REGION Network 65: Transfer P&P Gague R&R Job Interface [Hipot & Thickness Loading][Right]
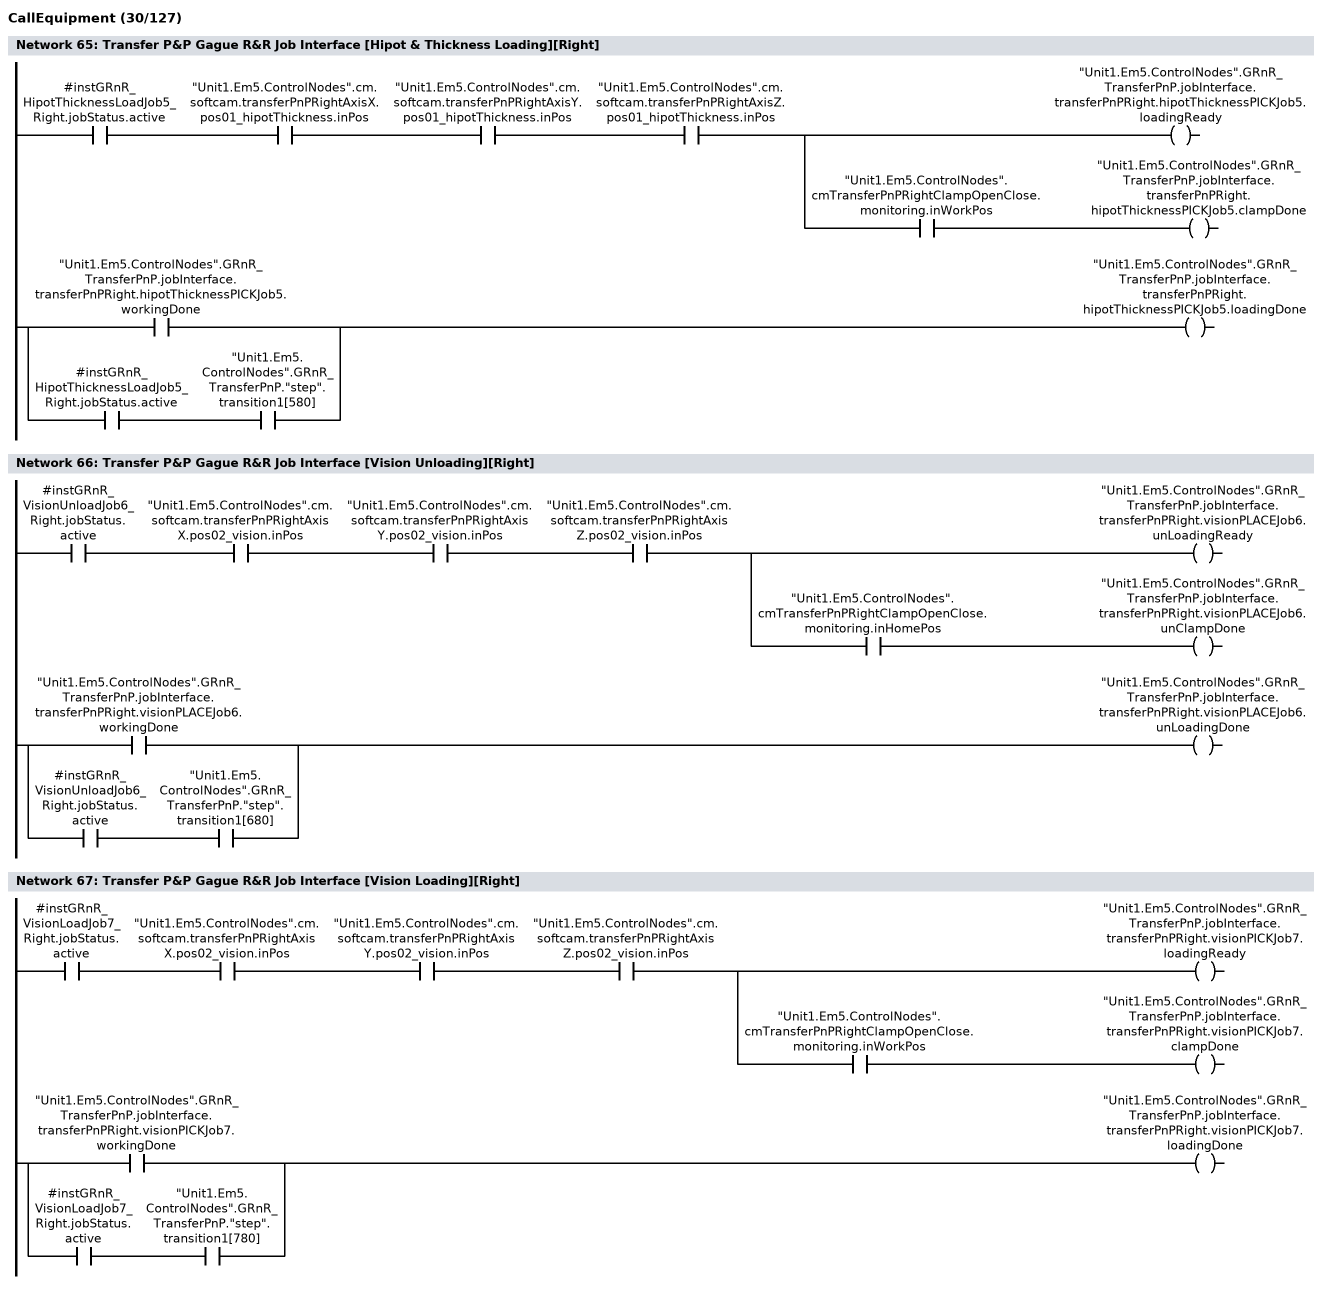
   RUNG wire#powerrail
      Contact( #instGRnR_HipotThicknessLoadJob5_Right.jobStatus.active )
      Contact( "Unit1.Em5.ControlNodes".cm.softcam.transferPnPRightAxisX.pos01_hipotThickness.inPos )
      Contact( "Unit1.Em5.ControlNodes".cm.softcam.transferPnPRightAxisY.pos01_hipotThickness.inPos )
      Contact( "Unit1.Em5.ControlNodes".cm.softcam.transferPnPRightAxisZ.pos01_hipotThickness.inPos )
      wire#w1
      Coil( "Unit1.Em5.ControlNodes".GRnR_TransferPnP.jobInterface.transferPnPRight.hipotThicknessPICKJob5.loadingReady )
   END_RUNG
   RUNG wire#w1
      Contact( "Unit1.Em5.ControlNodes".cmTransferPnPRightClampOpenClose.monitoring.inWorkPos )
      Coil( "Unit1.Em5.ControlNodes".GRnR_TransferPnP.jobInterface.transferPnPRight.hipotThicknessPICKJob5.clampDone )
   END_RUNG
   RUNG wire#powerrail
      Contact( "Unit1.Em5.ControlNodes".GRnR_TransferPnP.jobInterface.transferPnPRight.hipotThicknessPICKJob5.workingDone )
      wire#w2
      Coil( "Unit1.Em5.ControlNodes".GRnR_TransferPnP.jobInterface.transferPnPRight.hipotThicknessPICKJob5.loadingDone )
   END_RUNG
   RUNG wire#powerrail
      Contact( #instGRnR_HipotThicknessLoadJob5_Right.jobStatus.active )
      Contact( "Unit1.Em5.ControlNodes".GRnR_TransferPnP."step".transition1[580] )
   END_RUNG wire#w2
   // the same network as SCL:
   "Unit1.Em5.ControlNodes".GRnR_TransferPnP.jobInterface.transferPnPRight.hipotThicknessPICKJob5.loadingReady := #instGRnR_HipotThicknessLoadJob5_Right.jobStatus.active AND "Unit1.Em5.ControlNodes".cm.softcam.transferPnPRightAxisX.pos01_hipotThickness.inPos AND "Unit1.Em5.ControlNodes".cm.softcam.transferPnPRightAxisY.pos01_hipotThickness.inPos AND "Unit1.Em5.ControlNodes".cm.softcam.transferPnPRightAxisZ.pos01_hipotThickness.inPos;
   "Unit1.Em5.ControlNodes".GRnR_TransferPnP.jobInterface.transferPnPRight.hipotThicknessPICKJob5.clampDone := "Unit1.Em5.ControlNodes".GRnR_TransferPnP.jobInterface.transferPnPRight.hipotThicknessPICKJob5.loadingReady AND "Unit1.Em5.ControlNodes".cmTransferPnPRightClampOpenClose.monitoring.inWorkPos;
   "Unit1.Em5.ControlNodes".GRnR_TransferPnP.jobInterface.transferPnPRight.hipotThicknessPICKJob5.loadingDone := "Unit1.Em5.ControlNodes".GRnR_TransferPnP.jobInterface.transferPnPRight.hipotThicknessPICKJob5.workingDone OR (#instGRnR_HipotThicknessLoadJob5_Right.jobStatus.active AND "Unit1.Em5.ControlNodes".GRnR_TransferPnP."step".transition1[580]);
END_REGION

REGION Network 66: Transfer P&P Gague R&R Job Interface [Vision Unloading][Right]
   RUNG wire#powerrail
      Contact( #instGRnR_VisionUnloadJob6_Right.jobStatus.active )
      Contact( "Unit1.Em5.ControlNodes".cm.softcam.transferPnPRightAxisX.pos02_vision.inPos )
      Contact( "Unit1.Em5.ControlNodes".cm.softcam.transferPnPRightAxisY.pos02_vision.inPos )
      Contact( "Unit1.Em5.ControlNodes".cm.softcam.transferPnPRightAxisZ.pos02_vision.inPos )
      wire#w1
      Coil( "Unit1.Em5.ControlNodes".GRnR_TransferPnP.jobInterface.transferPnPRight.visionPLACEJob6.unLoadingReady )
   END_RUNG
   RUNG wire#w1
      Contact( "Unit1.Em5.ControlNodes".cmTransferPnPRightClampOpenClose.monitoring.inHomePos )
      Coil( "Unit1.Em5.ControlNodes".GRnR_TransferPnP.jobInterface.transferPnPRight.visionPLACEJob6.unClampDone )
   END_RUNG
   RUNG wire#powerrail
      Contact( "Unit1.Em5.ControlNodes".GRnR_TransferPnP.jobInterface.transferPnPRight.visionPLACEJob6.workingDone )
      wire#w2
      Coil( "Unit1.Em5.ControlNodes".GRnR_TransferPnP.jobInterface.transferPnPRight.visionPLACEJob6.unLoadingDone )
   END_RUNG
   RUNG wire#powerrail
      Contact( #instGRnR_VisionUnloadJob6_Right.jobStatus.active )
      Contact( "Unit1.Em5.ControlNodes".GRnR_TransferPnP."step".transition1[680] )
   END_RUNG wire#w2
   // the same network as SCL:
   "Unit1.Em5.ControlNodes".GRnR_TransferPnP.jobInterface.transferPnPRight.visionPLACEJob6.unLoadingReady := #instGRnR_VisionUnloadJob6_Right.jobStatus.active AND "Unit1.Em5.ControlNodes".cm.softcam.transferPnPRightAxisX.pos02_vision.inPos AND "Unit1.Em5.ControlNodes".cm.softcam.transferPnPRightAxisY.pos02_vision.inPos AND "Unit1.Em5.ControlNodes".cm.softcam.transferPnPRightAxisZ.pos02_vision.inPos;
   "Unit1.Em5.ControlNodes".GRnR_TransferPnP.jobInterface.transferPnPRight.visionPLACEJob6.unClampDone := "Unit1.Em5.ControlNodes".GRnR_TransferPnP.jobInterface.transferPnPRight.visionPLACEJob6.unLoadingReady AND "Unit1.Em5.ControlNodes".cmTransferPnPRightClampOpenClose.monitoring.inHomePos;
   "Unit1.Em5.ControlNodes".GRnR_TransferPnP.jobInterface.transferPnPRight.visionPLACEJob6.unLoadingDone := "Unit1.Em5.ControlNodes".GRnR_TransferPnP.jobInterface.transferPnPRight.visionPLACEJob6.workingDone OR (#instGRnR_VisionUnloadJob6_Right.jobStatus.active AND "Unit1.Em5.ControlNodes".GRnR_TransferPnP."step".transition1[680]);
END_REGION

REGION Network 67: Transfer P&P Gague R&R Job Interface [Vision Loading][Right]
   RUNG wire#powerrail
      Contact( #instGRnR_VisionLoadJob7_Right.jobStatus.active )
      Contact( "Unit1.Em5.ControlNodes".cm.softcam.transferPnPRightAxisX.pos02_vision.inPos )
      Contact( "Unit1.Em5.ControlNodes".cm.softcam.transferPnPRightAxisY.pos02_vision.inPos )
      Contact( "Unit1.Em5.ControlNodes".cm.softcam.transferPnPRightAxisZ.pos02_vision.inPos )
      wire#w1
      Coil( "Unit1.Em5.ControlNodes".GRnR_TransferPnP.jobInterface.transferPnPRight.visionPICKJob7.loadingReady )
   END_RUNG
   RUNG wire#w1
      Contact( "Unit1.Em5.ControlNodes".cmTransferPnPRightClampOpenClose.monitoring.inWorkPos )
      Coil( "Unit1.Em5.ControlNodes".GRnR_TransferPnP.jobInterface.transferPnPRight.visionPICKJob7.clampDone )
   END_RUNG
   RUNG wire#powerrail
      Contact( "Unit1.Em5.ControlNodes".GRnR_TransferPnP.jobInterface.transferPnPRight.visionPICKJob7.workingDone )
      wire#w2
      Coil( "Unit1.Em5.ControlNodes".GRnR_TransferPnP.jobInterface.transferPnPRight.visionPICKJob7.loadingDone )
   END_RUNG
   RUNG wire#powerrail
      Contact( #instGRnR_VisionLoadJob7_Right.jobStatus.active )
      Contact( "Unit1.Em5.ControlNodes".GRnR_TransferPnP."step".transition1[780] )
   END_RUNG wire#w2
   // the same network as SCL:
   "Unit1.Em5.ControlNodes".GRnR_TransferPnP.jobInterface.transferPnPRight.visionPICKJob7.loadingReady := #instGRnR_VisionLoadJob7_Right.jobStatus.active AND "Unit1.Em5.ControlNodes".cm.softcam.transferPnPRightAxisX.pos02_vision.inPos AND "Unit1.Em5.ControlNodes".cm.softcam.transferPnPRightAxisY.pos02_vision.inPos AND "Unit1.Em5.ControlNodes".cm.softcam.transferPnPRightAxisZ.pos02_vision.inPos;
   "Unit1.Em5.ControlNodes".GRnR_TransferPnP.jobInterface.transferPnPRight.visionPICKJob7.clampDone := "Unit1.Em5.ControlNodes".GRnR_TransferPnP.jobInterface.transferPnPRight.visionPICKJob7.loadingReady AND "Unit1.Em5.ControlNodes".cmTransferPnPRightClampOpenClose.monitoring.inWorkPos;
   "Unit1.Em5.ControlNodes".GRnR_TransferPnP.jobInterface.transferPnPRight.visionPICKJob7.loadingDone := "Unit1.Em5.ControlNodes".GRnR_TransferPnP.jobInterface.transferPnPRight.visionPICKJob7.workingDone OR (#instGRnR_VisionLoadJob7_Right.jobStatus.active AND "Unit1.Em5.ControlNodes".GRnR_TransferPnP."step".transition1[780]);
END_REGION

REGION Network 68: Transfer P&P Gague R&R Job Interface [Weight Check Unloading][Right]
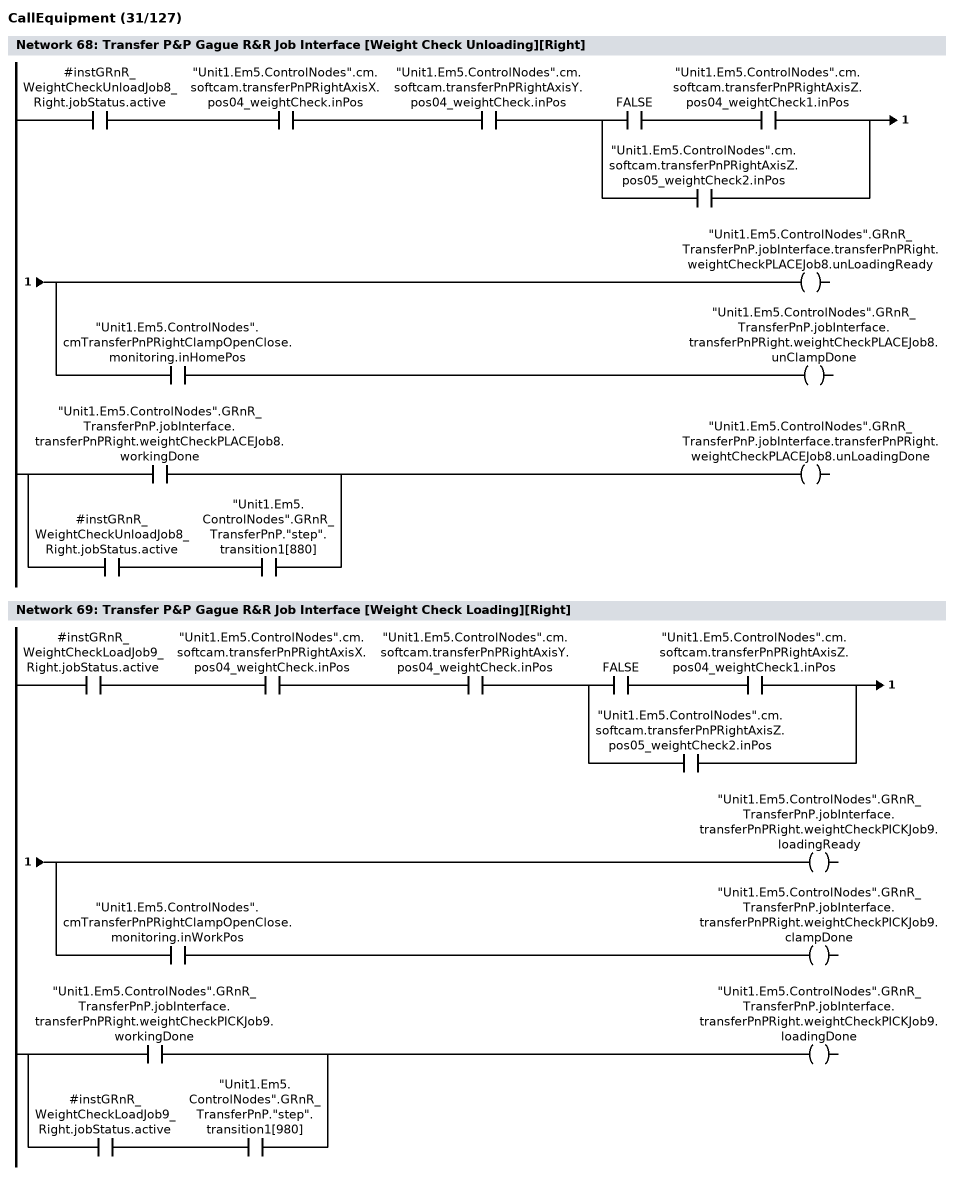
   RUNG wire#powerrail
      Contact( #instGRnR_WeightCheckUnloadJob8_Right.jobStatus.active )
      Contact( "Unit1.Em5.ControlNodes".cm.softcam.transferPnPRightAxisX.pos04_weightCheck.inPos )
      Contact( "Unit1.Em5.ControlNodes".cm.softcam.transferPnPRightAxisY.pos04_weightCheck.inPos )
      wire#w1
      Contact( FALSE )
      Contact( "Unit1.Em5.ControlNodes".cm.softcam.transferPnPRightAxisZ.pos04_weightCheck1.inPos )
      wire#w2
      Coil( "Unit1.Em5.ControlNodes".GRnR_TransferPnP.jobInterface.transferPnPRight.weightCheckPLACEJob8.unLoadingReady )
   END_RUNG
   RUNG wire#w1
      Contact( "Unit1.Em5.ControlNodes".cm.softcam.transferPnPRightAxisZ.pos05_weightCheck2.inPos )
   END_RUNG wire#w2
   RUNG wire#w2
      Contact( "Unit1.Em5.ControlNodes".cmTransferPnPRightClampOpenClose.monitoring.inHomePos )
      Coil( "Unit1.Em5.ControlNodes".GRnR_TransferPnP.jobInterface.transferPnPRight.weightCheckPLACEJob8.unClampDone )
   END_RUNG
   RUNG wire#powerrail
      Contact( "Unit1.Em5.ControlNodes".GRnR_TransferPnP.jobInterface.transferPnPRight.weightCheckPLACEJob8.workingDone )
      wire#w3
      Coil( "Unit1.Em5.ControlNodes".GRnR_TransferPnP.jobInterface.transferPnPRight.weightCheckPLACEJob8.unLoadingDone )
   END_RUNG
   RUNG wire#powerrail
      Contact( #instGRnR_WeightCheckUnloadJob8_Right.jobStatus.active )
      Contact( "Unit1.Em5.ControlNodes".GRnR_TransferPnP."step".transition1[880] )
   END_RUNG wire#w3
   // the same network as SCL:
   "Unit1.Em5.ControlNodes".GRnR_TransferPnP.jobInterface.transferPnPRight.weightCheckPLACEJob8.unLoadingReady := #instGRnR_WeightCheckUnloadJob8_Right.jobStatus.active AND "Unit1.Em5.ControlNodes".cm.softcam.transferPnPRightAxisX.pos04_weightCheck.inPos AND "Unit1.Em5.ControlNodes".cm.softcam.transferPnPRightAxisY.pos04_weightCheck.inPos AND ((FALSE AND "Unit1.Em5.ControlNodes".cm.softcam.transferPnPRightAxisZ.pos04_weightCheck1.inPos) OR "Unit1.Em5.ControlNodes".cm.softcam.transferPnPRightAxisZ.pos05_weightCheck2.inPos);
   "Unit1.Em5.ControlNodes".GRnR_TransferPnP.jobInterface.transferPnPRight.weightCheckPLACEJob8.unClampDone := "Unit1.Em5.ControlNodes".GRnR_TransferPnP.jobInterface.transferPnPRight.weightCheckPLACEJob8.unLoadingReady AND "Unit1.Em5.ControlNodes".cmTransferPnPRightClampOpenClose.monitoring.inHomePos;
   "Unit1.Em5.ControlNodes".GRnR_TransferPnP.jobInterface.transferPnPRight.weightCheckPLACEJob8.unLoadingDone := "Unit1.Em5.ControlNodes".GRnR_TransferPnP.jobInterface.transferPnPRight.weightCheckPLACEJob8.workingDone OR (#instGRnR_WeightCheckUnloadJob8_Right.jobStatus.active AND "Unit1.Em5.ControlNodes".GRnR_TransferPnP."step".transition1[880]);
END_REGION

REGION Network 69: Transfer P&P Gague R&R Job Interface [Weight Check Loading][Right]
   RUNG wire#powerrail
      Contact( #instGRnR_WeightCheckLoadJob9_Right.jobStatus.active )
      Contact( "Unit1.Em5.ControlNodes".cm.softcam.transferPnPRightAxisX.pos04_weightCheck.inPos )
      Contact( "Unit1.Em5.ControlNodes".cm.softcam.transferPnPRightAxisY.pos04_weightCheck.inPos )
      wire#w1
      Contact( FALSE )
      Contact( "Unit1.Em5.ControlNodes".cm.softcam.transferPnPRightAxisZ.pos04_weightCheck1.inPos )
      wire#w2
      Coil( "Unit1.Em5.ControlNodes".GRnR_TransferPnP.jobInterface.transferPnPRight.weightCheckPICKJob9.loadingReady )
   END_RUNG
   RUNG wire#w1
      Contact( "Unit1.Em5.ControlNodes".cm.softcam.transferPnPRightAxisZ.pos05_weightCheck2.inPos )
   END_RUNG wire#w2
   RUNG wire#w2
      Contact( "Unit1.Em5.ControlNodes".cmTransferPnPRightClampOpenClose.monitoring.inWorkPos )
      Coil( "Unit1.Em5.ControlNodes".GRnR_TransferPnP.jobInterface.transferPnPRight.weightCheckPICKJob9.clampDone )
   END_RUNG
   RUNG wire#powerrail
      Contact( "Unit1.Em5.ControlNodes".GRnR_TransferPnP.jobInterface.transferPnPRight.weightCheckPICKJob9.workingDone )
      wire#w3
      Coil( "Unit1.Em5.ControlNodes".GRnR_TransferPnP.jobInterface.transferPnPRight.weightCheckPICKJob9.loadingDone )
   END_RUNG
   RUNG wire#powerrail
      Contact( #instGRnR_WeightCheckLoadJob9_Right.jobStatus.active )
      Contact( "Unit1.Em5.ControlNodes".GRnR_TransferPnP."step".transition1[980] )
   END_RUNG wire#w3
   // the same network as SCL:
   "Unit1.Em5.ControlNodes".GRnR_TransferPnP.jobInterface.transferPnPRight.weightCheckPICKJob9.loadingReady := #instGRnR_WeightCheckLoadJob9_Right.jobStatus.active AND "Unit1.Em5.ControlNodes".cm.softcam.transferPnPRightAxisX.pos04_weightCheck.inPos AND "Unit1.Em5.ControlNodes".cm.softcam.transferPnPRightAxisY.pos04_weightCheck.inPos AND ((FALSE AND "Unit1.Em5.ControlNodes".cm.softcam.transferPnPRightAxisZ.pos04_weightCheck1.inPos) OR "Unit1.Em5.ControlNodes".cm.softcam.transferPnPRightAxisZ.pos05_weightCheck2.inPos);
   "Unit1.Em5.ControlNodes".GRnR_TransferPnP.jobInterface.transferPnPRight.weightCheckPICKJob9.clampDone := "Unit1.Em5.ControlNodes".GRnR_TransferPnP.jobInterface.transferPnPRight.weightCheckPICKJob9.loadingReady AND "Unit1.Em5.ControlNodes".cmTransferPnPRightClampOpenClose.monitoring.inWorkPos;
   "Unit1.Em5.ControlNodes".GRnR_TransferPnP.jobInterface.transferPnPRight.weightCheckPICKJob9.loadingDone := "Unit1.Em5.ControlNodes".GRnR_TransferPnP.jobInterface.transferPnPRight.weightCheckPICKJob9.workingDone OR (#instGRnR_WeightCheckLoadJob9_Right.jobStatus.active AND "Unit1.Em5.ControlNodes".GRnR_TransferPnP."step".transition1[980]);
END_REGION

REGION Network 70: Transfer P&P Gague R&R Job Interface Working Done [Side Tape → Hipot & Thickness]
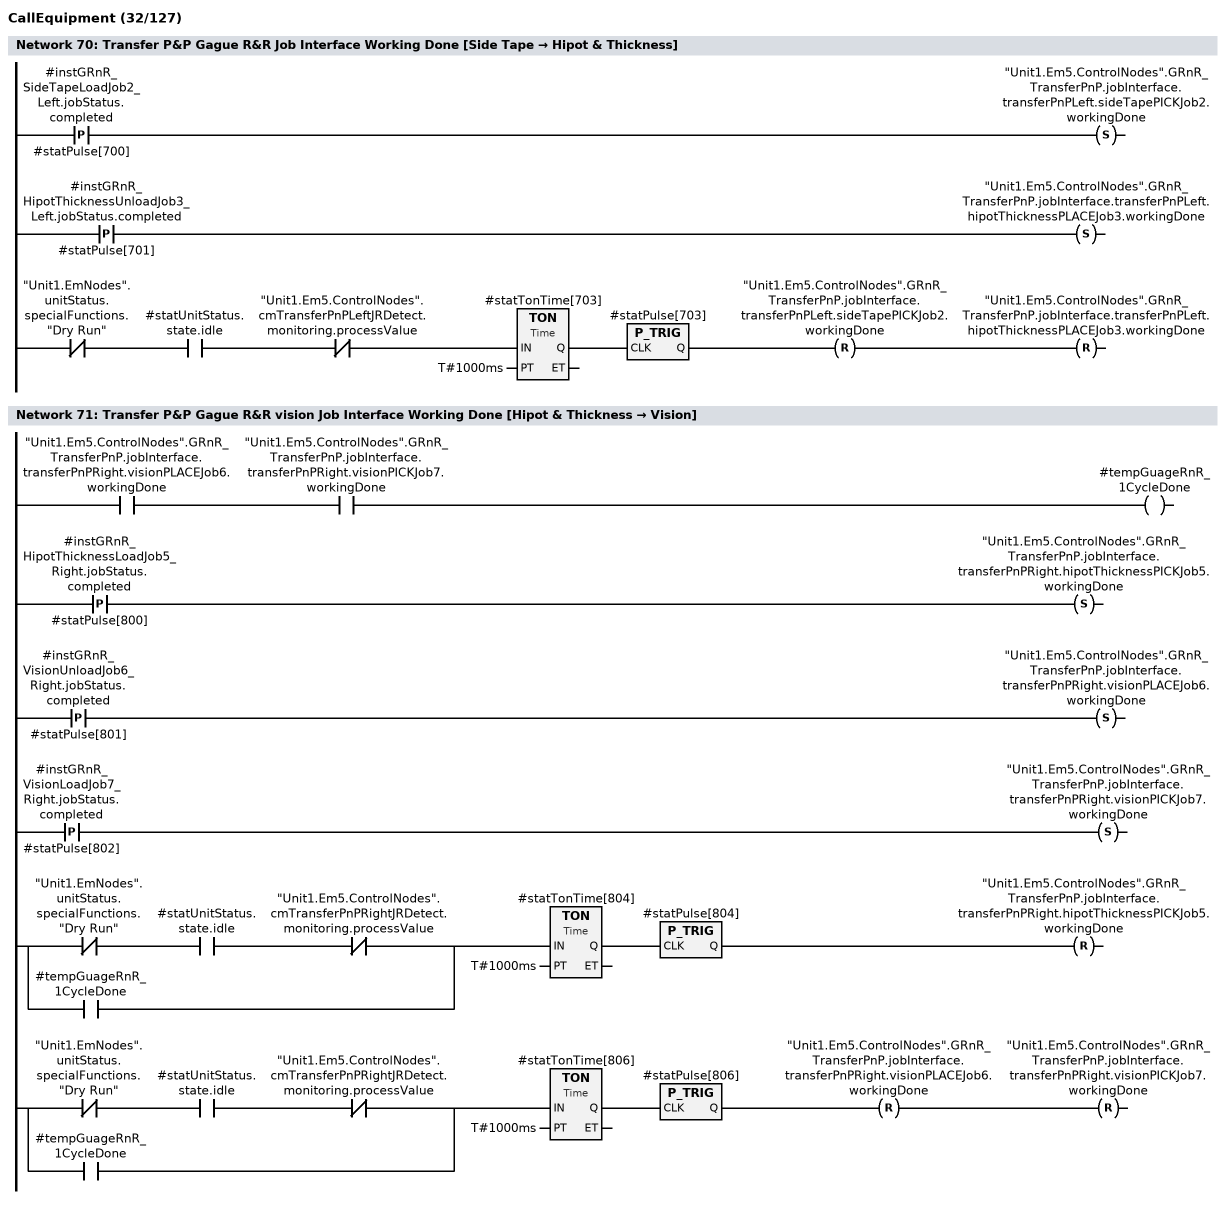
   RUNG wire#powerrail
      P_Contact(operand := #instGRnR_SideTapeLoadJob2_Left.jobStatus.completed, bit := #statPulse[700])
      S_Coil( "Unit1.Em5.ControlNodes".GRnR_TransferPnP.jobInterface.transferPnPLeft.sideTapePICKJob2.workingDone )
   END_RUNG
   RUNG wire#powerrail
      P_Contact(operand := #instGRnR_HipotThicknessUnloadJob3_Left.jobStatus.completed, bit := #statPulse[701])
      S_Coil( "Unit1.Em5.ControlNodes".GRnR_TransferPnP.jobInterface.transferPnPLeft.hipotThicknessPLACEJob3.workingDone )
   END_RUNG
   RUNG wire#powerrail
      I_Contact( "Unit1.EmNodes".unitStatus.specialFunctions."Dry Run" )
      Contact( #statUnitStatus.state.idle )
      I_Contact( "Unit1.Em5.ControlNodes".cmTransferPnPLeftJRDetect.monitoring.processValue )
      { S7_Templates := "time_type := Time" } #statTonTime[703].TON(pt := T#1000ms, et =>)
      P_Trig( #statPulse[703] )
      R_Coil( "Unit1.Em5.ControlNodes".GRnR_TransferPnP.jobInterface.transferPnPLeft.sideTapePICKJob2.workingDone )
      R_Coil( "Unit1.Em5.ControlNodes".GRnR_TransferPnP.jobInterface.transferPnPLeft.hipotThicknessPLACEJob3.workingDone )
   END_RUNG
   // the same network as SCL:
   #_w1 := #instGRnR_SideTapeLoadJob2_Left.jobStatus.completed AND NOT #statPulse[700];   // rising edge of #instGRnR_SideTapeLoadJob2_Left.jobStatus.completed
   #statPulse[700] := #instGRnR_SideTapeLoadJob2_Left.jobStatus.completed;
   IF #_w1 THEN
       "Unit1.Em5.ControlNodes".GRnR_TransferPnP.jobInterface.transferPnPLeft.sideTapePICKJob2.workingDone := TRUE;
   END_IF;
   #_w2 := #instGRnR_HipotThicknessUnloadJob3_Left.jobStatus.completed AND NOT #statPulse[701];   // rising edge of #instGRnR_HipotThicknessUnloadJob3_Left.jobStatus.completed
   #statPulse[701] := #instGRnR_HipotThicknessUnloadJob3_Left.jobStatus.completed;
   IF #_w2 THEN
       "Unit1.Em5.ControlNodes".GRnR_TransferPnP.jobInterface.transferPnPLeft.hipotThicknessPLACEJob3.workingDone := TRUE;
   END_IF;
   #statTonTime[703].TON(IN := NOT "Unit1.EmNodes".unitStatus.specialFunctions."Dry Run" AND #statUnitStatus.state.idle AND NOT "Unit1.Em5.ControlNodes".cmTransferPnPLeftJRDetect.monitoring.processValue,
                         PT := T#1000ms);
   #_w3 := #statTonTime[703].Q AND NOT #statPulse[703];   // rising edge
   #statPulse[703] := #statTonTime[703].Q;
   IF #_w3 THEN
       "Unit1.Em5.ControlNodes".GRnR_TransferPnP.jobInterface.transferPnPLeft.sideTapePICKJob2.workingDone := FALSE;
       "Unit1.Em5.ControlNodes".GRnR_TransferPnP.jobInterface.transferPnPLeft.hipotThicknessPLACEJob3.workingDone := FALSE;
   END_IF;
END_REGION

REGION Network 71: Transfer P&P Gague R&R vision Job Interface Working Done [Hipot & Thickness → Vision]
   RUNG wire#powerrail
      Contact( "Unit1.Em5.ControlNodes".GRnR_TransferPnP.jobInterface.transferPnPRight.visionPLACEJob6.workingDone )
      Contact( "Unit1.Em5.ControlNodes".GRnR_TransferPnP.jobInterface.transferPnPRight.visionPICKJob7.workingDone )
      Coil( #tempGuageRnR_1CycleDone )
   END_RUNG
   RUNG wire#powerrail
      P_Contact(operand := #instGRnR_HipotThicknessLoadJob5_Right.jobStatus.completed, bit := #statPulse[800])
      S_Coil( "Unit1.Em5.ControlNodes".GRnR_TransferPnP.jobInterface.transferPnPRight.hipotThicknessPICKJob5.workingDone )
   END_RUNG
   RUNG wire#powerrail
      P_Contact(operand := #instGRnR_VisionUnloadJob6_Right.jobStatus.completed, bit := #statPulse[801])
      S_Coil( "Unit1.Em5.ControlNodes".GRnR_TransferPnP.jobInterface.transferPnPRight.visionPLACEJob6.workingDone )
   END_RUNG
   RUNG wire#powerrail
      P_Contact(operand := #instGRnR_VisionLoadJob7_Right.jobStatus.completed, bit := #statPulse[802])
      S_Coil( "Unit1.Em5.ControlNodes".GRnR_TransferPnP.jobInterface.transferPnPRight.visionPICKJob7.workingDone )
   END_RUNG
   RUNG wire#powerrail
      I_Contact( "Unit1.EmNodes".unitStatus.specialFunctions."Dry Run" )
      Contact( #statUnitStatus.state.idle )
      I_Contact( "Unit1.Em5.ControlNodes".cmTransferPnPRightJRDetect.monitoring.processValue )
      wire#w1
      { S7_Templates := "time_type := Time" } #statTonTime[804].TON(pt := T#1000ms, et =>)
      P_Trig( #statPulse[804] )
      R_Coil( "Unit1.Em5.ControlNodes".GRnR_TransferPnP.jobInterface.transferPnPRight.hipotThicknessPICKJob5.workingDone )
   END_RUNG
   RUNG wire#powerrail
      Contact( #tempGuageRnR_1CycleDone )
   END_RUNG wire#w1
   RUNG wire#powerrail
      I_Contact( "Unit1.EmNodes".unitStatus.specialFunctions."Dry Run" )
      Contact( #statUnitStatus.state.idle )
      I_Contact( "Unit1.Em5.ControlNodes".cmTransferPnPRightJRDetect.monitoring.processValue )
      wire#w2
      { S7_Templates := "time_type := Time" } #statTonTime[806].TON(pt := T#1000ms, et =>)
      P_Trig( #statPulse[806] )
      R_Coil( "Unit1.Em5.ControlNodes".GRnR_TransferPnP.jobInterface.transferPnPRight.visionPLACEJob6.workingDone )
      R_Coil( "Unit1.Em5.ControlNodes".GRnR_TransferPnP.jobInterface.transferPnPRight.visionPICKJob7.workingDone )
   END_RUNG
   RUNG wire#powerrail
      Contact( #tempGuageRnR_1CycleDone )
   END_RUNG wire#w2
   // the same network as SCL:
   #tempGuageRnR_1CycleDone := "Unit1.Em5.ControlNodes".GRnR_TransferPnP.jobInterface.transferPnPRight.visionPLACEJob6.workingDone AND "Unit1.Em5.ControlNodes".GRnR_TransferPnP.jobInterface.transferPnPRight.visionPICKJob7.workingDone;
   #_w1 := #instGRnR_HipotThicknessLoadJob5_Right.jobStatus.completed AND NOT #statPulse[800];   // rising edge of #instGRnR_HipotThicknessLoadJob5_Right.jobStatus.completed
   #statPulse[800] := #instGRnR_HipotThicknessLoadJob5_Right.jobStatus.completed;
   IF #_w1 THEN
       "Unit1.Em5.ControlNodes".GRnR_TransferPnP.jobInterface.transferPnPRight.hipotThicknessPICKJob5.workingDone := TRUE;
   END_IF;
   #_w2 := #instGRnR_VisionUnloadJob6_Right.jobStatus.completed AND NOT #statPulse[801];   // rising edge of #instGRnR_VisionUnloadJob6_Right.jobStatus.completed
   #statPulse[801] := #instGRnR_VisionUnloadJob6_Right.jobStatus.completed;
   IF #_w2 THEN
       "Unit1.Em5.ControlNodes".GRnR_TransferPnP.jobInterface.transferPnPRight.visionPLACEJob6.workingDone := TRUE;
   END_IF;
   #_w3 := #instGRnR_VisionLoadJob7_Right.jobStatus.completed AND NOT #statPulse[802];   // rising edge of #instGRnR_VisionLoadJob7_Right.jobStatus.completed
   #statPulse[802] := #instGRnR_VisionLoadJob7_Right.jobStatus.completed;
   IF #_w3 THEN
       "Unit1.Em5.ControlNodes".GRnR_TransferPnP.jobInterface.transferPnPRight.visionPICKJob7.workingDone := TRUE;
   END_IF;
   #statTonTime[804].TON(IN := (NOT "Unit1.EmNodes".unitStatus.specialFunctions."Dry Run" AND #statUnitStatus.state.idle AND NOT "Unit1.Em5.ControlNodes".cmTransferPnPRightJRDetect.monitoring.processValue) OR #tempGuageRnR_1CycleDone,
                         PT := T#1000ms);
   #_w4 := #statTonTime[804].Q AND NOT #statPulse[804];   // rising edge
   #statPulse[804] := #statTonTime[804].Q;
   IF #_w4 THEN
       "Unit1.Em5.ControlNodes".GRnR_TransferPnP.jobInterface.transferPnPRight.hipotThicknessPICKJob5.workingDone := FALSE;
   END_IF;
   #statTonTime[806].TON(IN := (NOT "Unit1.EmNodes".unitStatus.specialFunctions."Dry Run" AND #statUnitStatus.state.idle AND NOT "Unit1.Em5.ControlNodes".cmTransferPnPRightJRDetect.monitoring.processValue) OR #tempGuageRnR_1CycleDone,
                         PT := T#1000ms);
   #_w5 := #statTonTime[806].Q AND NOT #statPulse[806];   // rising edge
   #statPulse[806] := #statTonTime[806].Q;
   IF #_w5 THEN
       "Unit1.Em5.ControlNodes".GRnR_TransferPnP.jobInterface.transferPnPRight.visionPLACEJob6.workingDone := FALSE;
       "Unit1.Em5.ControlNodes".GRnR_TransferPnP.jobInterface.transferPnPRight.visionPICKJob7.workingDone := FALSE;
   END_IF;
END_REGION

REGION Network 72: Transfer P&P Gague R&R Job Interface Working Done [Vision → Weight Check]
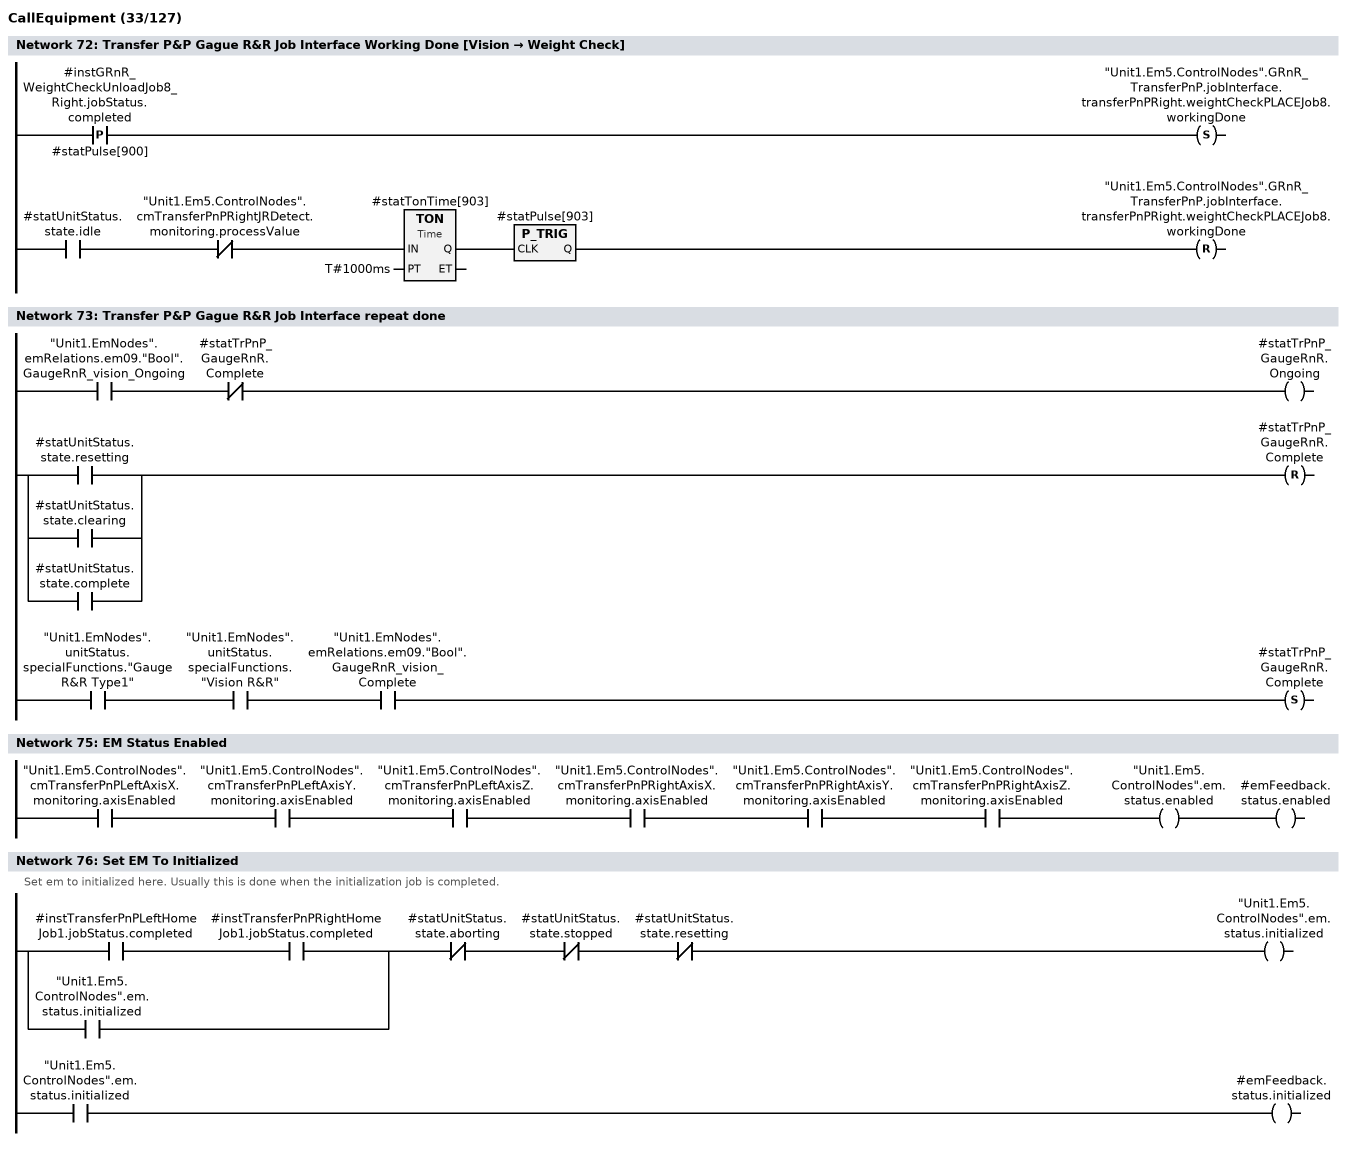
   RUNG wire#powerrail
      P_Contact(operand := #instGRnR_WeightCheckUnloadJob8_Right.jobStatus.completed, bit := #statPulse[900])
      S_Coil( "Unit1.Em5.ControlNodes".GRnR_TransferPnP.jobInterface.transferPnPRight.weightCheckPLACEJob8.workingDone )
   END_RUNG
   RUNG wire#powerrail
      Contact( #statUnitStatus.state.idle )
      I_Contact( "Unit1.Em5.ControlNodes".cmTransferPnPRightJRDetect.monitoring.processValue )
      { S7_Templates := "time_type := Time" } #statTonTime[903].TON(pt := T#1000ms, et =>)
      P_Trig( #statPulse[903] )
      R_Coil( "Unit1.Em5.ControlNodes".GRnR_TransferPnP.jobInterface.transferPnPRight.weightCheckPLACEJob8.workingDone )
   END_RUNG
   // the same network as SCL:
   #_w1 := #instGRnR_WeightCheckUnloadJob8_Right.jobStatus.completed AND NOT #statPulse[900];   // rising edge of #instGRnR_WeightCheckUnloadJob8_Right.jobStatus.completed
   #statPulse[900] := #instGRnR_WeightCheckUnloadJob8_Right.jobStatus.completed;
   IF #_w1 THEN
       "Unit1.Em5.ControlNodes".GRnR_TransferPnP.jobInterface.transferPnPRight.weightCheckPLACEJob8.workingDone := TRUE;
   END_IF;
   #statTonTime[903].TON(IN := #statUnitStatus.state.idle AND NOT "Unit1.Em5.ControlNodes".cmTransferPnPRightJRDetect.monitoring.processValue,
                         PT := T#1000ms);
   #_w2 := #statTonTime[903].Q AND NOT #statPulse[903];   // rising edge
   #statPulse[903] := #statTonTime[903].Q;
   IF #_w2 THEN
       "Unit1.Em5.ControlNodes".GRnR_TransferPnP.jobInterface.transferPnPRight.weightCheckPLACEJob8.workingDone := FALSE;
   END_IF;
END_REGION

REGION Network 73: Transfer P&P Gague R&R Job Interface repeat done
   RUNG wire#powerrail
      Contact( "Unit1.EmNodes".emRelations.em09."Bool".GaugeRnR_vision_Ongoing )
      I_Contact( #statTrPnP_GaugeRnR.Complete )
      Coil( #statTrPnP_GaugeRnR.Ongoing )
   END_RUNG
   RUNG wire#powerrail
      Contact( #statUnitStatus.state.resetting )
      wire#w1
      R_Coil( #statTrPnP_GaugeRnR.Complete )
   END_RUNG
   RUNG wire#powerrail
      Contact( #statUnitStatus.state.clearing )
   END_RUNG wire#w1
   RUNG wire#powerrail
      Contact( #statUnitStatus.state.complete )
   END_RUNG wire#w1
   RUNG wire#powerrail
      Contact( "Unit1.EmNodes".unitStatus.specialFunctions."Gauge R&R Type1" )
      Contact( "Unit1.EmNodes".unitStatus.specialFunctions."Vision R&R" )
      Contact( "Unit1.EmNodes".emRelations.em09."Bool".GaugeRnR_vision_Complete )
      S_Coil( #statTrPnP_GaugeRnR.Complete )
   END_RUNG
   // the same network as SCL:
   #statTrPnP_GaugeRnR.Ongoing := "Unit1.EmNodes".emRelations.em09."Bool".GaugeRnR_vision_Ongoing AND NOT #statTrPnP_GaugeRnR.Complete;
   IF #statUnitStatus.state.resetting OR #statUnitStatus.state.clearing OR #statUnitStatus.state.complete THEN
       #statTrPnP_GaugeRnR.Complete := FALSE;
   END_IF;
   IF "Unit1.EmNodes".unitStatus.specialFunctions."Gauge R&R Type1" AND "Unit1.EmNodes".unitStatus.specialFunctions."Vision R&R" AND "Unit1.EmNodes".emRelations.em09."Bool".GaugeRnR_vision_Complete THEN
       #statTrPnP_GaugeRnR.Complete := TRUE;
   END_IF;
END_REGION

REGION Network 75: EM Status Enabled
   RUNG wire#powerrail
      Contact( "Unit1.Em5.ControlNodes".cmTransferPnPLeftAxisX.monitoring.axisEnabled )
      Contact( "Unit1.Em5.ControlNodes".cmTransferPnPLeftAxisY.monitoring.axisEnabled )
      Contact( "Unit1.Em5.ControlNodes".cmTransferPnPLeftAxisZ.monitoring.axisEnabled )
      Contact( "Unit1.Em5.ControlNodes".cmTransferPnPRightAxisX.monitoring.axisEnabled )
      Contact( "Unit1.Em5.ControlNodes".cmTransferPnPRightAxisY.monitoring.axisEnabled )
      Contact( "Unit1.Em5.ControlNodes".cmTransferPnPRightAxisZ.monitoring.axisEnabled )
      Coil( "Unit1.Em5.ControlNodes".em.status.enabled )
      Coil( #emFeedback.status.enabled )
   END_RUNG
   // the same network as SCL:
   "Unit1.Em5.ControlNodes".em.status.enabled := "Unit1.Em5.ControlNodes".cmTransferPnPLeftAxisX.monitoring.axisEnabled AND "Unit1.Em5.ControlNodes".cmTransferPnPLeftAxisY.monitoring.axisEnabled AND "Unit1.Em5.ControlNodes".cmTransferPnPLeftAxisZ.monitoring.axisEnabled AND "Unit1.Em5.ControlNodes".cmTransferPnPRightAxisX.monitoring.axisEnabled AND "Unit1.Em5.ControlNodes".cmTransferPnPRightAxisY.monitoring.axisEnabled AND "Unit1.Em5.ControlNodes".cmTransferPnPRightAxisZ.monitoring.axisEnabled;
   #emFeedback.status.enabled := "Unit1.Em5.ControlNodes".em.status.enabled;
END_REGION

REGION Network 76: Set EM To Initialized
   // Set em to initialized here. Usually this is done when the initialization job is completed.
   RUNG wire#powerrail
      Contact( #instTransferPnPLeftHomeJob1.jobStatus.completed )
      Contact( #instTransferPnPRightHomeJob1.jobStatus.completed )
      wire#w1
      I_Contact( #statUnitStatus.state.aborting )
      I_Contact( #statUnitStatus.state.stopped )
      I_Contact( #statUnitStatus.state.resetting )
      Coil( "Unit1.Em5.ControlNodes".em.status.initialized )
   END_RUNG
   RUNG wire#powerrail
      Contact( "Unit1.Em5.ControlNodes".em.status.initialized )
   END_RUNG wire#w1
   RUNG wire#powerrail
      Contact( "Unit1.Em5.ControlNodes".em.status.initialized )
      Coil( #emFeedback.status.initialized )
   END_RUNG
   // the same network as SCL:
   "Unit1.Em5.ControlNodes".em.status.initialized := ((#instTransferPnPLeftHomeJob1.jobStatus.completed AND #instTransferPnPRightHomeJob1.jobStatus.completed) OR "Unit1.Em5.ControlNodes".em.status.initialized) AND NOT #statUnitStatus.state.aborting AND NOT #statUnitStatus.state.stopped AND NOT #statUnitStatus.state.resetting;
   #emFeedback.status.initialized := "Unit1.Em5.ControlNodes".em.status.initialized;
END_REGION

REGION Network 77: EM Status Homed
   // DefaultPosPartDetect : TR PnP Right has a Part, and no where to go
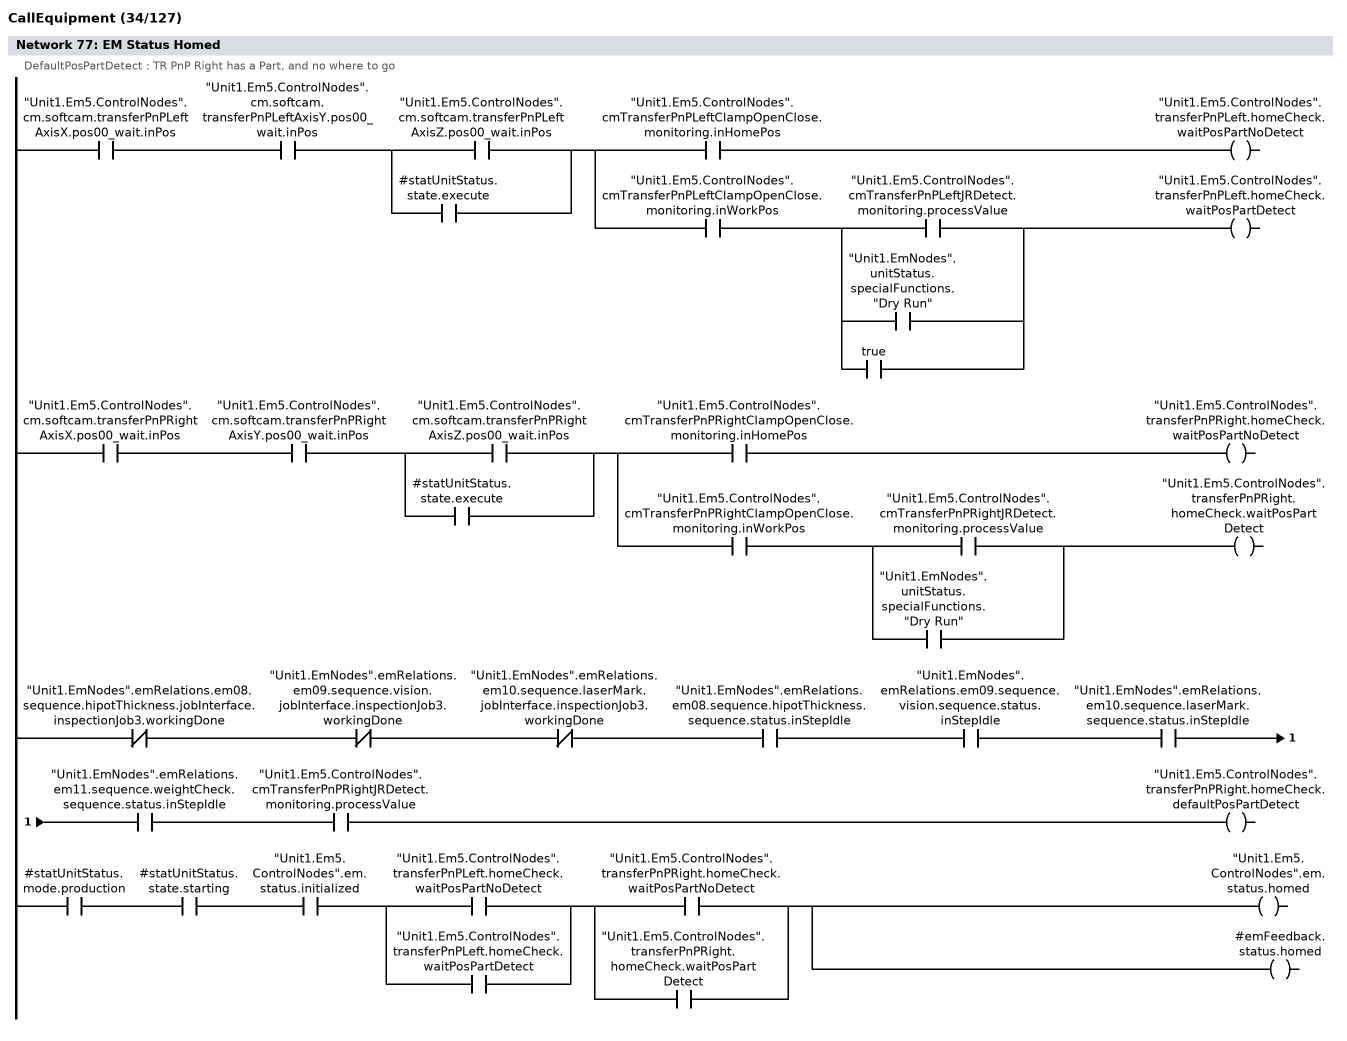
   RUNG wire#powerrail
      Contact( "Unit1.Em5.ControlNodes".cm.softcam.transferPnPLeftAxisX.pos00_wait.inPos )
      Contact( "Unit1.Em5.ControlNodes".cm.softcam.transferPnPLeftAxisY.pos00_wait.inPos )
      wire#w1
      Contact( "Unit1.Em5.ControlNodes".cm.softcam.transferPnPLeftAxisZ.pos00_wait.inPos )
      wire#w2
      Contact( "Unit1.Em5.ControlNodes".cmTransferPnPLeftClampOpenClose.monitoring.inHomePos )
      Coil( "Unit1.Em5.ControlNodes".transferPnPLeft.homeCheck.waitPosPartNoDetect )
   END_RUNG
   RUNG wire#w1
      Contact( #statUnitStatus.state.execute )
   END_RUNG wire#w2
   RUNG wire#w2
      Contact( "Unit1.Em5.ControlNodes".cmTransferPnPLeftClampOpenClose.monitoring.inWorkPos )
      wire#w3
      Contact( "Unit1.Em5.ControlNodes".cmTransferPnPLeftJRDetect.monitoring.processValue )
      wire#w4
      Coil( "Unit1.Em5.ControlNodes".transferPnPLeft.homeCheck.waitPosPartDetect )
   END_RUNG
   RUNG wire#w3
      Contact( "Unit1.EmNodes".unitStatus.specialFunctions."Dry Run" )
   END_RUNG wire#w4
   RUNG wire#w3
      Contact( true )
   END_RUNG wire#w4
   RUNG wire#powerrail
      Contact( "Unit1.Em5.ControlNodes".cm.softcam.transferPnPRightAxisX.pos00_wait.inPos )
      Contact( "Unit1.Em5.ControlNodes".cm.softcam.transferPnPRightAxisY.pos00_wait.inPos )
      wire#w5
      Contact( "Unit1.Em5.ControlNodes".cm.softcam.transferPnPRightAxisZ.pos00_wait.inPos )
      wire#w6
      Contact( "Unit1.Em5.ControlNodes".cmTransferPnPRightClampOpenClose.monitoring.inHomePos )
      Coil( "Unit1.Em5.ControlNodes".transferPnPRight.homeCheck.waitPosPartNoDetect )
   END_RUNG
   RUNG wire#w5
      Contact( #statUnitStatus.state.execute )
   END_RUNG wire#w6
   RUNG wire#w6
      Contact( "Unit1.Em5.ControlNodes".cmTransferPnPRightClampOpenClose.monitoring.inWorkPos )
      wire#w7
      Contact( "Unit1.Em5.ControlNodes".cmTransferPnPRightJRDetect.monitoring.processValue )
      wire#w8
      Coil( "Unit1.Em5.ControlNodes".transferPnPRight.homeCheck.waitPosPartDetect )
   END_RUNG
   RUNG wire#w7
      Contact( "Unit1.EmNodes".unitStatus.specialFunctions."Dry Run" )
   END_RUNG wire#w8
   RUNG wire#powerrail
      I_Contact( "Unit1.EmNodes".emRelations.em08.sequence.hipotThickness.jobInterface.inspectionJob3.workingDone )
      I_Contact( "Unit1.EmNodes".emRelations.em09.sequence.vision.jobInterface.inspectionJob3.workingDone )
      I_Contact( "Unit1.EmNodes".emRelations.em10.sequence.laserMark.jobInterface.inspectionJob3.workingDone )
      Contact( "Unit1.EmNodes".emRelations.em08.sequence.hipotThickness.sequence.status.inStepIdle )
      Contact( "Unit1.EmNodes".emRelations.em09.sequence.vision.sequence.status.inStepIdle )
      Contact( "Unit1.EmNodes".emRelations.em10.sequence.laserMark.sequence.status.inStepIdle )
      Contact( "Unit1.EmNodes".emRelations.em11.sequence.weightCheck.sequence.status.inStepIdle )
      Contact( "Unit1.Em5.ControlNodes".cmTransferPnPRightJRDetect.monitoring.processValue )
      Coil( "Unit1.Em5.ControlNodes".transferPnPRight.homeCheck.defaultPosPartDetect )
   END_RUNG
   RUNG wire#powerrail
      Contact( #statUnitStatus.mode.production )
      Contact( #statUnitStatus.state.starting )
      Contact( "Unit1.Em5.ControlNodes".em.status.initialized )
      wire#w9
      Contact( "Unit1.Em5.ControlNodes".transferPnPLeft.homeCheck.waitPosPartNoDetect )
      wire#w10
      Contact( "Unit1.Em5.ControlNodes".transferPnPRight.homeCheck.waitPosPartNoDetect )
      wire#w11
      Coil( "Unit1.Em5.ControlNodes".em.status.homed )
   END_RUNG
   RUNG wire#w9
      Contact( "Unit1.Em5.ControlNodes".transferPnPLeft.homeCheck.waitPosPartDetect )
   END_RUNG wire#w10
   RUNG wire#w10
      Contact( "Unit1.Em5.ControlNodes".transferPnPRight.homeCheck.waitPosPartDetect )
   END_RUNG wire#w11
   RUNG wire#w11
      Coil( #emFeedback.status.homed )
   END_RUNG
   // the same network as SCL:
   #_w1 := "Unit1.Em5.ControlNodes".cm.softcam.transferPnPLeftAxisX.pos00_wait.inPos AND "Unit1.Em5.ControlNodes".cm.softcam.transferPnPLeftAxisY.pos00_wait.inPos AND ("Unit1.Em5.ControlNodes".cm.softcam.transferPnPLeftAxisZ.pos00_wait.inPos OR #statUnitStatus.state.execute);
   "Unit1.Em5.ControlNodes".transferPnPLeft.homeCheck.waitPosPartNoDetect := #_w1 AND "Unit1.Em5.ControlNodes".cmTransferPnPLeftClampOpenClose.monitoring.inHomePos;
   "Unit1.Em5.ControlNodes".transferPnPLeft.homeCheck.waitPosPartDetect := #_w1 AND "Unit1.Em5.ControlNodes".cmTransferPnPLeftClampOpenClose.monitoring.inWorkPos AND ("Unit1.Em5.ControlNodes".cmTransferPnPLeftJRDetect.monitoring.processValue OR "Unit1.EmNodes".unitStatus.specialFunctions."Dry Run" OR true);
   #_w2 := "Unit1.Em5.ControlNodes".cm.softcam.transferPnPRightAxisX.pos00_wait.inPos AND "Unit1.Em5.ControlNodes".cm.softcam.transferPnPRightAxisY.pos00_wait.inPos AND ("Unit1.Em5.ControlNodes".cm.softcam.transferPnPRightAxisZ.pos00_wait.inPos OR #statUnitStatus.state.execute);
   "Unit1.Em5.ControlNodes".transferPnPRight.homeCheck.waitPosPartNoDetect := #_w2 AND "Unit1.Em5.ControlNodes".cmTransferPnPRightClampOpenClose.monitoring.inHomePos;
   "Unit1.Em5.ControlNodes".transferPnPRight.homeCheck.waitPosPartDetect := #_w2 AND "Unit1.Em5.ControlNodes".cmTransferPnPRightClampOpenClose.monitoring.inWorkPos AND ("Unit1.Em5.ControlNodes".cmTransferPnPRightJRDetect.monitoring.processValue OR "Unit1.EmNodes".unitStatus.specialFunctions."Dry Run");
   "Unit1.Em5.ControlNodes".transferPnPRight.homeCheck.defaultPosPartDetect := NOT "Unit1.EmNodes".emRelations.em08.sequence.hipotThickness.jobInterface.inspectionJob3.workingDone AND NOT "Unit1.EmNodes".emRelations.em09.sequence.vision.jobInterface.inspectionJob3.workingDone AND NOT "Unit1.EmNodes".emRelations.em10.sequence.laserMark.jobInterface.inspectionJob3.workingDone AND "Unit1.EmNodes".emRelations.em08.sequence.hipotThickness.sequence.status.inStepIdle AND "Unit1.EmNodes".emRelations.em09.sequence.vision.sequence.status.inStepIdle AND "Unit1.EmNodes".emRelations.em10.sequence.laserMark.sequence.status.inStepIdle AND "Unit1.EmNodes".emRelations.em11.sequence.weightCheck.sequence.status.inStepIdle AND "Unit1.Em5.ControlNodes".cmTransferPnPRightJRDetect.monitoring.processValue;
   "Unit1.Em5.ControlNodes".em.status.homed := #statUnitStatus.mode.production AND #statUnitStatus.state.starting AND "Unit1.Em5.ControlNodes".em.status.initialized AND ("Unit1.Em5.ControlNodes".transferPnPLeft.homeCheck.waitPosPartNoDetect OR "Unit1.Em5.ControlNodes".transferPnPLeft.homeCheck.waitPosPartDetect) AND ("Unit1.Em5.ControlNodes".transferPnPRight.homeCheck.waitPosPartNoDetect OR "Unit1.Em5.ControlNodes".transferPnPRight.homeCheck.waitPosPartDetect);
   #emFeedback.status.homed := "Unit1.Em5.ControlNodes".em.status.homed;
END_REGION

REGION Network 78: Transfer P&P Left Position Check
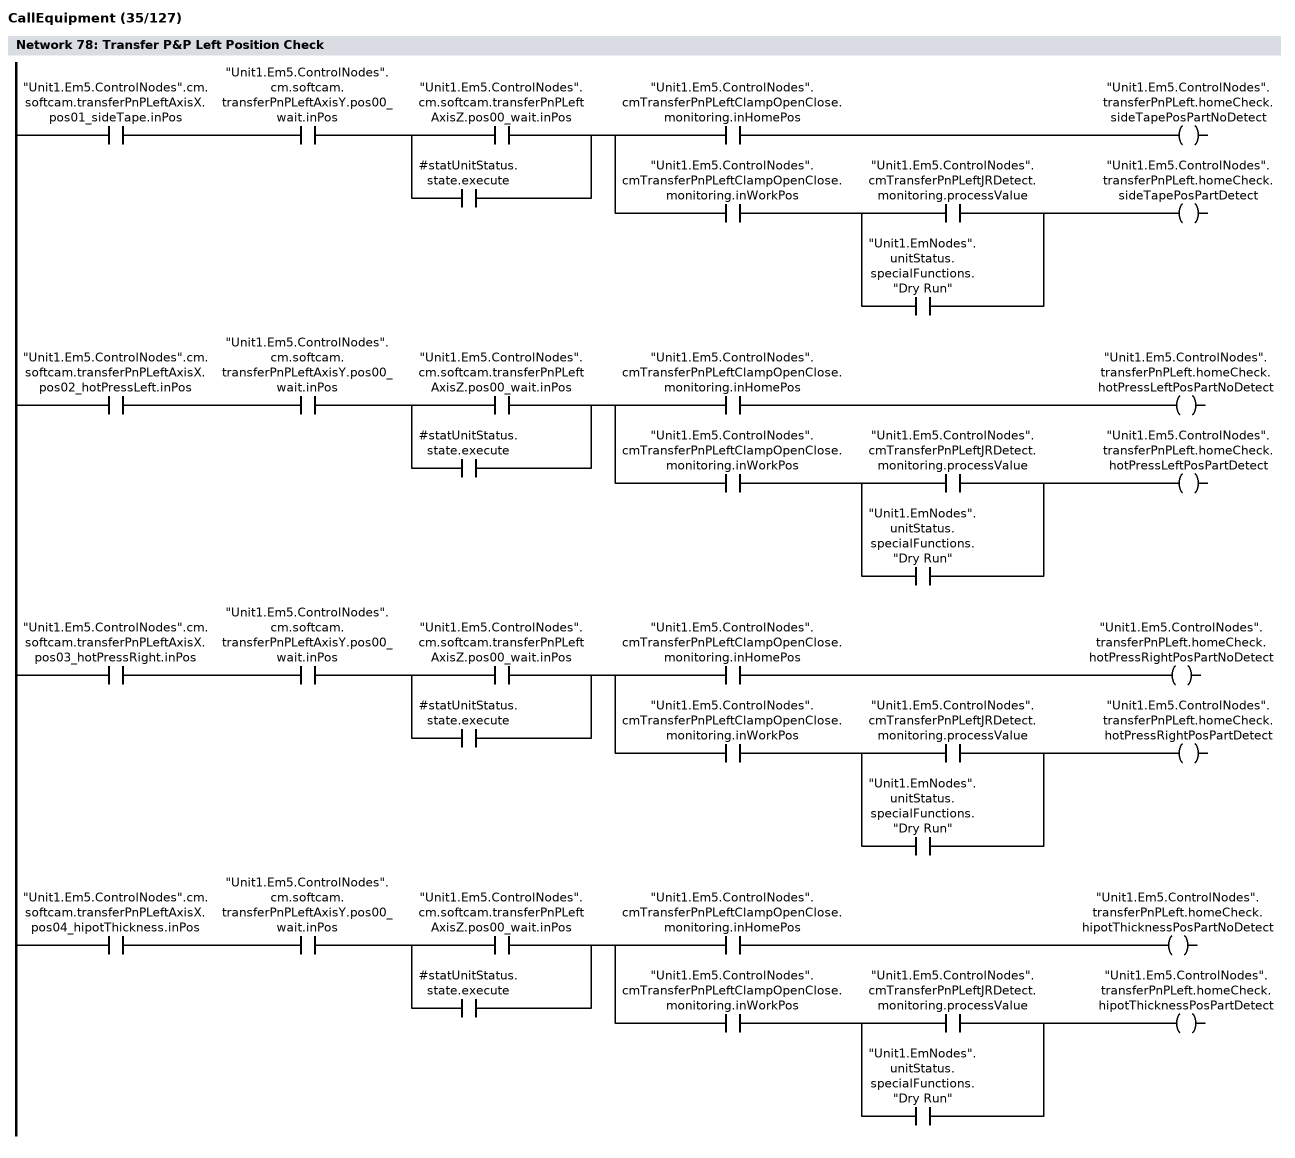
   RUNG wire#powerrail
      Contact( "Unit1.Em5.ControlNodes".cm.softcam.transferPnPLeftAxisX.pos01_sideTape.inPos )
      Contact( "Unit1.Em5.ControlNodes".cm.softcam.transferPnPLeftAxisY.pos00_wait.inPos )
      wire#w1
      Contact( "Unit1.Em5.ControlNodes".cm.softcam.transferPnPLeftAxisZ.pos00_wait.inPos )
      wire#w2
      Contact( "Unit1.Em5.ControlNodes".cmTransferPnPLeftClampOpenClose.monitoring.inHomePos )
      Coil( "Unit1.Em5.ControlNodes".transferPnPLeft.homeCheck.sideTapePosPartNoDetect )
   END_RUNG
   RUNG wire#w1
      Contact( #statUnitStatus.state.execute )
   END_RUNG wire#w2
   RUNG wire#w2
      Contact( "Unit1.Em5.ControlNodes".cmTransferPnPLeftClampOpenClose.monitoring.inWorkPos )
      wire#w3
      Contact( "Unit1.Em5.ControlNodes".cmTransferPnPLeftJRDetect.monitoring.processValue )
      wire#w4
      Coil( "Unit1.Em5.ControlNodes".transferPnPLeft.homeCheck.sideTapePosPartDetect )
   END_RUNG
   RUNG wire#w3
      Contact( "Unit1.EmNodes".unitStatus.specialFunctions."Dry Run" )
   END_RUNG wire#w4
   RUNG wire#powerrail
      Contact( "Unit1.Em5.ControlNodes".cm.softcam.transferPnPLeftAxisX.pos02_hotPressLeft.inPos )
      Contact( "Unit1.Em5.ControlNodes".cm.softcam.transferPnPLeftAxisY.pos00_wait.inPos )
      wire#w5
      Contact( "Unit1.Em5.ControlNodes".cm.softcam.transferPnPLeftAxisZ.pos00_wait.inPos )
      wire#w6
      Contact( "Unit1.Em5.ControlNodes".cmTransferPnPLeftClampOpenClose.monitoring.inHomePos )
      Coil( "Unit1.Em5.ControlNodes".transferPnPLeft.homeCheck.hotPressLeftPosPartNoDetect )
   END_RUNG
   RUNG wire#w5
      Contact( #statUnitStatus.state.execute )
   END_RUNG wire#w6
   RUNG wire#w6
      Contact( "Unit1.Em5.ControlNodes".cmTransferPnPLeftClampOpenClose.monitoring.inWorkPos )
      wire#w7
      Contact( "Unit1.Em5.ControlNodes".cmTransferPnPLeftJRDetect.monitoring.processValue )
      wire#w8
      Coil( "Unit1.Em5.ControlNodes".transferPnPLeft.homeCheck.hotPressLeftPosPartDetect )
   END_RUNG
   RUNG wire#w7
      Contact( "Unit1.EmNodes".unitStatus.specialFunctions."Dry Run" )
   END_RUNG wire#w8
   RUNG wire#powerrail
      Contact( "Unit1.Em5.ControlNodes".cm.softcam.transferPnPLeftAxisX.pos03_hotPressRight.inPos )
      Contact( "Unit1.Em5.ControlNodes".cm.softcam.transferPnPLeftAxisY.pos00_wait.inPos )
      wire#w9
      Contact( "Unit1.Em5.ControlNodes".cm.softcam.transferPnPLeftAxisZ.pos00_wait.inPos )
      wire#w10
      Contact( "Unit1.Em5.ControlNodes".cmTransferPnPLeftClampOpenClose.monitoring.inHomePos )
      Coil( "Unit1.Em5.ControlNodes".transferPnPLeft.homeCheck.hotPressRightPosPartNoDetect )
   END_RUNG
   RUNG wire#w9
      Contact( #statUnitStatus.state.execute )
   END_RUNG wire#w10
   RUNG wire#w10
      Contact( "Unit1.Em5.ControlNodes".cmTransferPnPLeftClampOpenClose.monitoring.inWorkPos )
      wire#w11
      Contact( "Unit1.Em5.ControlNodes".cmTransferPnPLeftJRDetect.monitoring.processValue )
      wire#w12
      Coil( "Unit1.Em5.ControlNodes".transferPnPLeft.homeCheck.hotPressRightPosPartDetect )
   END_RUNG
   RUNG wire#w11
      Contact( "Unit1.EmNodes".unitStatus.specialFunctions."Dry Run" )
   END_RUNG wire#w12
   RUNG wire#powerrail
      Contact( "Unit1.Em5.ControlNodes".cm.softcam.transferPnPLeftAxisX.pos04_hipotThickness.inPos )
      Contact( "Unit1.Em5.ControlNodes".cm.softcam.transferPnPLeftAxisY.pos00_wait.inPos )
      wire#w13
      Contact( "Unit1.Em5.ControlNodes".cm.softcam.transferPnPLeftAxisZ.pos00_wait.inPos )
      wire#w14
      Contact( "Unit1.Em5.ControlNodes".cmTransferPnPLeftClampOpenClose.monitoring.inHomePos )
      Coil( "Unit1.Em5.ControlNodes".transferPnPLeft.homeCheck.hipotThicknessPosPartNoDetect )
   END_RUNG
   RUNG wire#w13
      Contact( #statUnitStatus.state.execute )
   END_RUNG wire#w14
   RUNG wire#w14
      Contact( "Unit1.Em5.ControlNodes".cmTransferPnPLeftClampOpenClose.monitoring.inWorkPos )
      wire#w15
      Contact( "Unit1.Em5.ControlNodes".cmTransferPnPLeftJRDetect.monitoring.processValue )
      wire#w16
      Coil( "Unit1.Em5.ControlNodes".transferPnPLeft.homeCheck.hipotThicknessPosPartDetect )
   END_RUNG
   RUNG wire#w15
      Contact( "Unit1.EmNodes".unitStatus.specialFunctions."Dry Run" )
   END_RUNG wire#w16
   // the same network as SCL:
   #_w1 := "Unit1.Em5.ControlNodes".cm.softcam.transferPnPLeftAxisX.pos01_sideTape.inPos AND "Unit1.Em5.ControlNodes".cm.softcam.transferPnPLeftAxisY.pos00_wait.inPos AND ("Unit1.Em5.ControlNodes".cm.softcam.transferPnPLeftAxisZ.pos00_wait.inPos OR #statUnitStatus.state.execute);
   "Unit1.Em5.ControlNodes".transferPnPLeft.homeCheck.sideTapePosPartNoDetect := #_w1 AND "Unit1.Em5.ControlNodes".cmTransferPnPLeftClampOpenClose.monitoring.inHomePos;
   "Unit1.Em5.ControlNodes".transferPnPLeft.homeCheck.sideTapePosPartDetect := #_w1 AND "Unit1.Em5.ControlNodes".cmTransferPnPLeftClampOpenClose.monitoring.inWorkPos AND ("Unit1.Em5.ControlNodes".cmTransferPnPLeftJRDetect.monitoring.processValue OR "Unit1.EmNodes".unitStatus.specialFunctions."Dry Run");
   #_w2 := "Unit1.Em5.ControlNodes".cm.softcam.transferPnPLeftAxisX.pos02_hotPressLeft.inPos AND "Unit1.Em5.ControlNodes".cm.softcam.transferPnPLeftAxisY.pos00_wait.inPos AND ("Unit1.Em5.ControlNodes".cm.softcam.transferPnPLeftAxisZ.pos00_wait.inPos OR #statUnitStatus.state.execute);
   "Unit1.Em5.ControlNodes".transferPnPLeft.homeCheck.hotPressLeftPosPartNoDetect := #_w2 AND "Unit1.Em5.ControlNodes".cmTransferPnPLeftClampOpenClose.monitoring.inHomePos;
   "Unit1.Em5.ControlNodes".transferPnPLeft.homeCheck.hotPressLeftPosPartDetect := #_w2 AND "Unit1.Em5.ControlNodes".cmTransferPnPLeftClampOpenClose.monitoring.inWorkPos AND ("Unit1.Em5.ControlNodes".cmTransferPnPLeftJRDetect.monitoring.processValue OR "Unit1.EmNodes".unitStatus.specialFunctions."Dry Run");
   #_w3 := "Unit1.Em5.ControlNodes".cm.softcam.transferPnPLeftAxisX.pos03_hotPressRight.inPos AND "Unit1.Em5.ControlNodes".cm.softcam.transferPnPLeftAxisY.pos00_wait.inPos AND ("Unit1.Em5.ControlNodes".cm.softcam.transferPnPLeftAxisZ.pos00_wait.inPos OR #statUnitStatus.state.execute);
   "Unit1.Em5.ControlNodes".transferPnPLeft.homeCheck.hotPressRightPosPartNoDetect := #_w3 AND "Unit1.Em5.ControlNodes".cmTransferPnPLeftClampOpenClose.monitoring.inHomePos;
   "Unit1.Em5.ControlNodes".transferPnPLeft.homeCheck.hotPressRightPosPartDetect := #_w3 AND "Unit1.Em5.ControlNodes".cmTransferPnPLeftClampOpenClose.monitoring.inWorkPos AND ("Unit1.Em5.ControlNodes".cmTransferPnPLeftJRDetect.monitoring.processValue OR "Unit1.EmNodes".unitStatus.specialFunctions."Dry Run");
   #_w4 := "Unit1.Em5.ControlNodes".cm.softcam.transferPnPLeftAxisX.pos04_hipotThickness.inPos AND "Unit1.Em5.ControlNodes".cm.softcam.transferPnPLeftAxisY.pos00_wait.inPos AND ("Unit1.Em5.ControlNodes".cm.softcam.transferPnPLeftAxisZ.pos00_wait.inPos OR #statUnitStatus.state.execute);
   "Unit1.Em5.ControlNodes".transferPnPLeft.homeCheck.hipotThicknessPosPartNoDetect := #_w4 AND "Unit1.Em5.ControlNodes".cmTransferPnPLeftClampOpenClose.monitoring.inHomePos;
   "Unit1.Em5.ControlNodes".transferPnPLeft.homeCheck.hipotThicknessPosPartDetect := #_w4 AND "Unit1.Em5.ControlNodes".cmTransferPnPLeftClampOpenClose.monitoring.inWorkPos AND ("Unit1.Em5.ControlNodes".cmTransferPnPLeftJRDetect.monitoring.processValue OR "Unit1.EmNodes".unitStatus.specialFunctions."Dry Run");
END_REGION

REGION Network 79: Transfer P&P Right Position Check
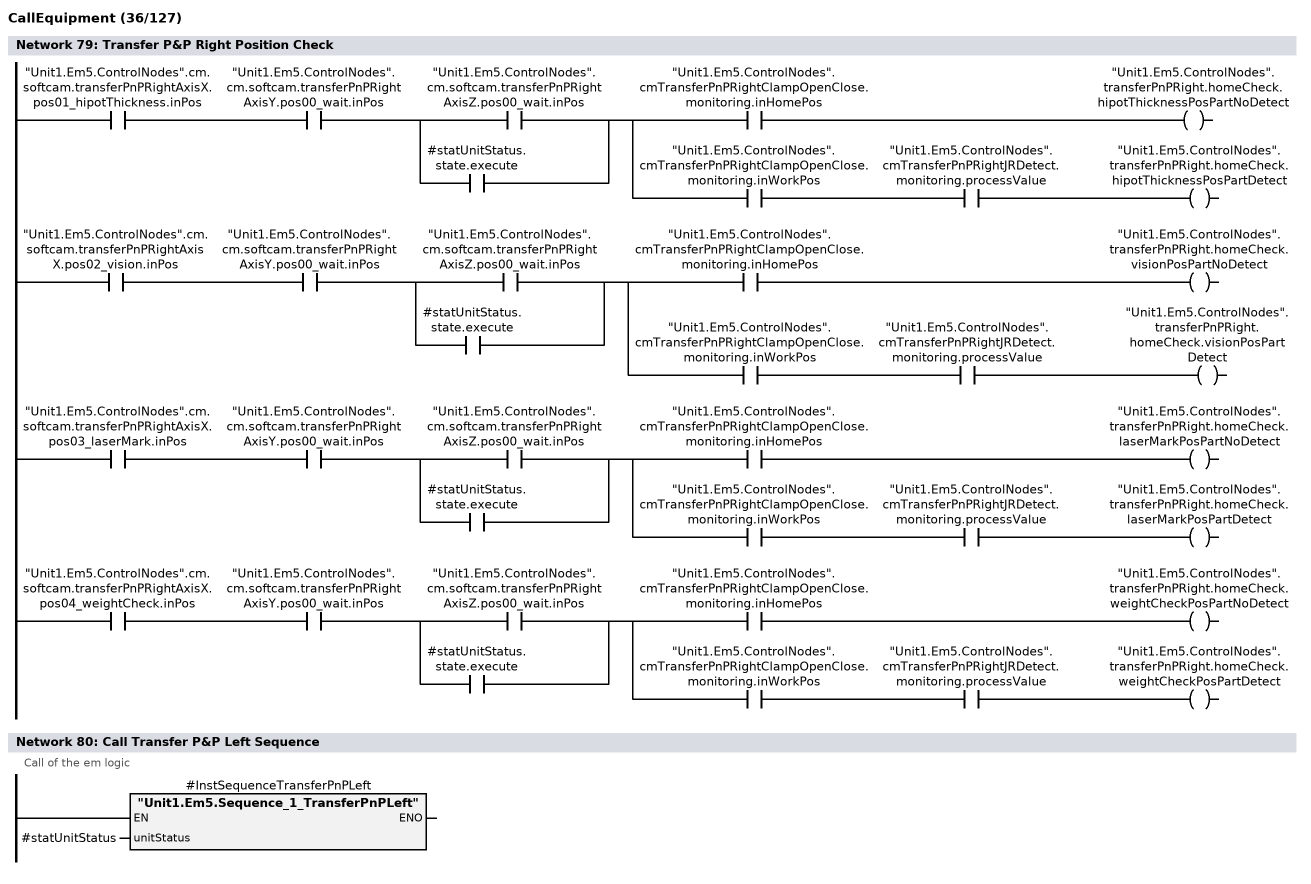
   RUNG wire#powerrail
      Contact( "Unit1.Em5.ControlNodes".cm.softcam.transferPnPRightAxisX.pos01_hipotThickness.inPos )
      Contact( "Unit1.Em5.ControlNodes".cm.softcam.transferPnPRightAxisY.pos00_wait.inPos )
      wire#w1
      Contact( "Unit1.Em5.ControlNodes".cm.softcam.transferPnPRightAxisZ.pos00_wait.inPos )
      wire#w2
      Contact( "Unit1.Em5.ControlNodes".cmTransferPnPRightClampOpenClose.monitoring.inHomePos )
      Coil( "Unit1.Em5.ControlNodes".transferPnPRight.homeCheck.hipotThicknessPosPartNoDetect )
   END_RUNG
   RUNG wire#w1
      Contact( #statUnitStatus.state.execute )
   END_RUNG wire#w2
   RUNG wire#w2
      Contact( "Unit1.Em5.ControlNodes".cmTransferPnPRightClampOpenClose.monitoring.inWorkPos )
      Contact( "Unit1.Em5.ControlNodes".cmTransferPnPRightJRDetect.monitoring.processValue )
      Coil( "Unit1.Em5.ControlNodes".transferPnPRight.homeCheck.hipotThicknessPosPartDetect )
   END_RUNG
   RUNG wire#powerrail
      Contact( "Unit1.Em5.ControlNodes".cm.softcam.transferPnPRightAxisX.pos02_vision.inPos )
      Contact( "Unit1.Em5.ControlNodes".cm.softcam.transferPnPRightAxisY.pos00_wait.inPos )
      wire#w3
      Contact( "Unit1.Em5.ControlNodes".cm.softcam.transferPnPRightAxisZ.pos00_wait.inPos )
      wire#w4
      Contact( "Unit1.Em5.ControlNodes".cmTransferPnPRightClampOpenClose.monitoring.inHomePos )
      Coil( "Unit1.Em5.ControlNodes".transferPnPRight.homeCheck.visionPosPartNoDetect )
   END_RUNG
   RUNG wire#w3
      Contact( #statUnitStatus.state.execute )
   END_RUNG wire#w4
   RUNG wire#w4
      Contact( "Unit1.Em5.ControlNodes".cmTransferPnPRightClampOpenClose.monitoring.inWorkPos )
      Contact( "Unit1.Em5.ControlNodes".cmTransferPnPRightJRDetect.monitoring.processValue )
      Coil( "Unit1.Em5.ControlNodes".transferPnPRight.homeCheck.visionPosPartDetect )
   END_RUNG
   RUNG wire#powerrail
      Contact( "Unit1.Em5.ControlNodes".cm.softcam.transferPnPRightAxisX.pos03_laserMark.inPos )
      Contact( "Unit1.Em5.ControlNodes".cm.softcam.transferPnPRightAxisY.pos00_wait.inPos )
      wire#w5
      Contact( "Unit1.Em5.ControlNodes".cm.softcam.transferPnPRightAxisZ.pos00_wait.inPos )
      wire#w6
      Contact( "Unit1.Em5.ControlNodes".cmTransferPnPRightClampOpenClose.monitoring.inHomePos )
      Coil( "Unit1.Em5.ControlNodes".transferPnPRight.homeCheck.laserMarkPosPartNoDetect )
   END_RUNG
   RUNG wire#w5
      Contact( #statUnitStatus.state.execute )
   END_RUNG wire#w6
   RUNG wire#w6
      Contact( "Unit1.Em5.ControlNodes".cmTransferPnPRightClampOpenClose.monitoring.inWorkPos )
      Contact( "Unit1.Em5.ControlNodes".cmTransferPnPRightJRDetect.monitoring.processValue )
      Coil( "Unit1.Em5.ControlNodes".transferPnPRight.homeCheck.laserMarkPosPartDetect )
   END_RUNG
   RUNG wire#powerrail
      Contact( "Unit1.Em5.ControlNodes".cm.softcam.transferPnPRightAxisX.pos04_weightCheck.inPos )
      Contact( "Unit1.Em5.ControlNodes".cm.softcam.transferPnPRightAxisY.pos00_wait.inPos )
      wire#w7
      Contact( "Unit1.Em5.ControlNodes".cm.softcam.transferPnPRightAxisZ.pos00_wait.inPos )
      wire#w8
      Contact( "Unit1.Em5.ControlNodes".cmTransferPnPRightClampOpenClose.monitoring.inHomePos )
      Coil( "Unit1.Em5.ControlNodes".transferPnPRight.homeCheck.weightCheckPosPartNoDetect )
   END_RUNG
   RUNG wire#w7
      Contact( #statUnitStatus.state.execute )
   END_RUNG wire#w8
   RUNG wire#w8
      Contact( "Unit1.Em5.ControlNodes".cmTransferPnPRightClampOpenClose.monitoring.inWorkPos )
      Contact( "Unit1.Em5.ControlNodes".cmTransferPnPRightJRDetect.monitoring.processValue )
      Coil( "Unit1.Em5.ControlNodes".transferPnPRight.homeCheck.weightCheckPosPartDetect )
   END_RUNG
   // the same network as SCL:
   #_w1 := "Unit1.Em5.ControlNodes".cm.softcam.transferPnPRightAxisX.pos01_hipotThickness.inPos AND "Unit1.Em5.ControlNodes".cm.softcam.transferPnPRightAxisY.pos00_wait.inPos AND ("Unit1.Em5.ControlNodes".cm.softcam.transferPnPRightAxisZ.pos00_wait.inPos OR #statUnitStatus.state.execute);
   "Unit1.Em5.ControlNodes".transferPnPRight.homeCheck.hipotThicknessPosPartNoDetect := #_w1 AND "Unit1.Em5.ControlNodes".cmTransferPnPRightClampOpenClose.monitoring.inHomePos;
   "Unit1.Em5.ControlNodes".transferPnPRight.homeCheck.hipotThicknessPosPartDetect := #_w1 AND "Unit1.Em5.ControlNodes".cmTransferPnPRightClampOpenClose.monitoring.inWorkPos AND "Unit1.Em5.ControlNodes".cmTransferPnPRightJRDetect.monitoring.processValue;
   #_w2 := "Unit1.Em5.ControlNodes".cm.softcam.transferPnPRightAxisX.pos02_vision.inPos AND "Unit1.Em5.ControlNodes".cm.softcam.transferPnPRightAxisY.pos00_wait.inPos AND ("Unit1.Em5.ControlNodes".cm.softcam.transferPnPRightAxisZ.pos00_wait.inPos OR #statUnitStatus.state.execute);
   "Unit1.Em5.ControlNodes".transferPnPRight.homeCheck.visionPosPartNoDetect := #_w2 AND "Unit1.Em5.ControlNodes".cmTransferPnPRightClampOpenClose.monitoring.inHomePos;
   "Unit1.Em5.ControlNodes".transferPnPRight.homeCheck.visionPosPartDetect := #_w2 AND "Unit1.Em5.ControlNodes".cmTransferPnPRightClampOpenClose.monitoring.inWorkPos AND "Unit1.Em5.ControlNodes".cmTransferPnPRightJRDetect.monitoring.processValue;
   #_w3 := "Unit1.Em5.ControlNodes".cm.softcam.transferPnPRightAxisX.pos03_laserMark.inPos AND "Unit1.Em5.ControlNodes".cm.softcam.transferPnPRightAxisY.pos00_wait.inPos AND ("Unit1.Em5.ControlNodes".cm.softcam.transferPnPRightAxisZ.pos00_wait.inPos OR #statUnitStatus.state.execute);
   "Unit1.Em5.ControlNodes".transferPnPRight.homeCheck.laserMarkPosPartNoDetect := #_w3 AND "Unit1.Em5.ControlNodes".cmTransferPnPRightClampOpenClose.monitoring.inHomePos;
   "Unit1.Em5.ControlNodes".transferPnPRight.homeCheck.laserMarkPosPartDetect := #_w3 AND "Unit1.Em5.ControlNodes".cmTransferPnPRightClampOpenClose.monitoring.inWorkPos AND "Unit1.Em5.ControlNodes".cmTransferPnPRightJRDetect.monitoring.processValue;
   #_w4 := "Unit1.Em5.ControlNodes".cm.softcam.transferPnPRightAxisX.pos04_weightCheck.inPos AND "Unit1.Em5.ControlNodes".cm.softcam.transferPnPRightAxisY.pos00_wait.inPos AND ("Unit1.Em5.ControlNodes".cm.softcam.transferPnPRightAxisZ.pos00_wait.inPos OR #statUnitStatus.state.execute);
   "Unit1.Em5.ControlNodes".transferPnPRight.homeCheck.weightCheckPosPartNoDetect := #_w4 AND "Unit1.Em5.ControlNodes".cmTransferPnPRightClampOpenClose.monitoring.inHomePos;
   "Unit1.Em5.ControlNodes".transferPnPRight.homeCheck.weightCheckPosPartDetect := #_w4 AND "Unit1.Em5.ControlNodes".cmTransferPnPRightClampOpenClose.monitoring.inWorkPos AND "Unit1.Em5.ControlNodes".cmTransferPnPRightJRDetect.monitoring.processValue;
END_REGION

REGION Network 80: Call Transfer P&P Left Sequence
   // Call of the em logic
   RUNG wire#powerrail
      #InstSequenceTransferPnPLeft(unitStatus := #statUnitStatus)
   END_RUNG
   // the same network as SCL:
   #InstSequenceTransferPnPLeft(unitStatus := #statUnitStatus);   // "Unit1.Em5.Sequence_1_TransferPnPLeft"
END_REGION

REGION Network 81: Transfer P&P Left Sequence Status
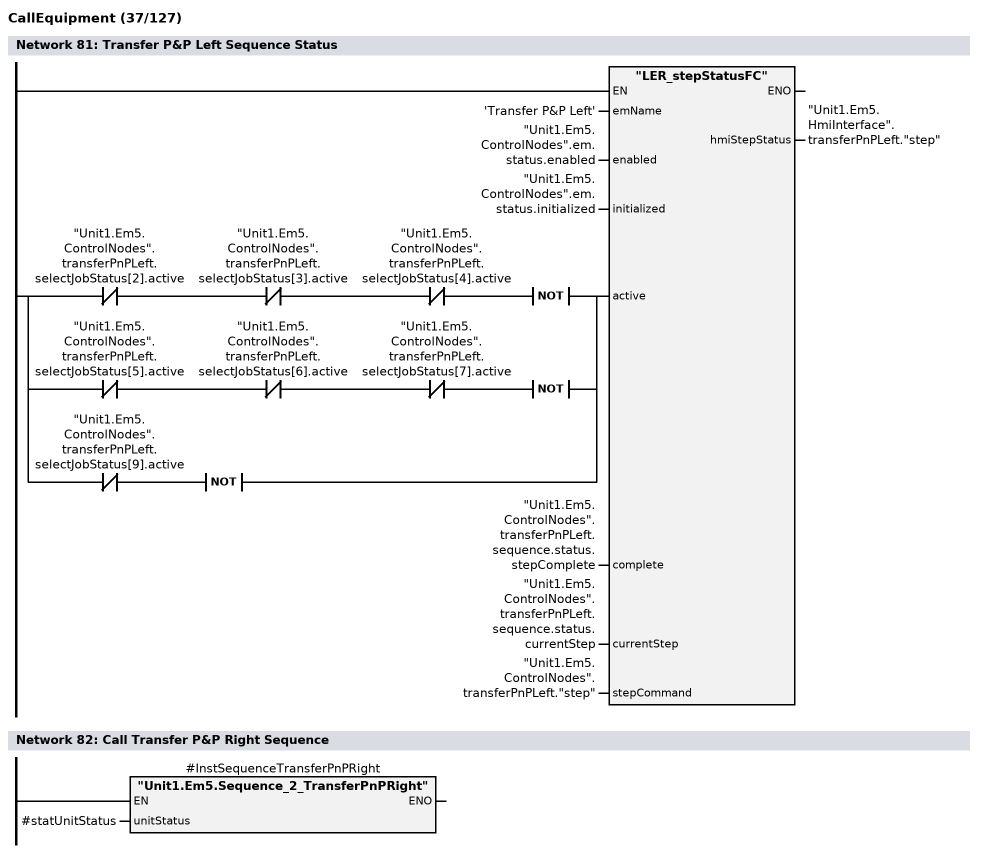
   RUNG wire#powerrail
      "LER_stepStatusFC"(active := wire#w1, emName := 'Transfer P&P Left', enabled := "Unit1.Em5.ControlNodes".em.status.enabled, initialized := "Unit1.Em5.ControlNodes".em.status.initialized, complete := "Unit1.Em5.ControlNodes".transferPnPLeft.sequence.status.stepComplete, currentStep := "Unit1.Em5.ControlNodes".transferPnPLeft.sequence.status.currentStep, stepCommand := "Unit1.Em5.ControlNodes".transferPnPLeft."step", hmiStepStatus => "Unit1.Em5.HmiInterface".transferPnPLeft."step")
   END_RUNG
   RUNG wire#powerrail
      I_Contact( "Unit1.Em5.ControlNodes".transferPnPLeft.selectJobStatus[2].active )
      I_Contact( "Unit1.Em5.ControlNodes".transferPnPLeft.selectJobStatus[3].active )
      I_Contact( "Unit1.Em5.ControlNodes".transferPnPLeft.selectJobStatus[4].active )
      Not()
   END_RUNG wire#w1
   RUNG wire#powerrail
      I_Contact( "Unit1.Em5.ControlNodes".transferPnPLeft.selectJobStatus[5].active )
      I_Contact( "Unit1.Em5.ControlNodes".transferPnPLeft.selectJobStatus[6].active )
      I_Contact( "Unit1.Em5.ControlNodes".transferPnPLeft.selectJobStatus[7].active )
      Not()
   END_RUNG wire#w1
   RUNG wire#powerrail
      I_Contact( "Unit1.Em5.ControlNodes".transferPnPLeft.selectJobStatus[9].active )
      Not()
   END_RUNG wire#w1
   // the same network as SCL:
   "LER_stepStatusFC"(emName := 'Transfer P&P Left',
                      enabled := "Unit1.Em5.ControlNodes".em.status.enabled,
                      initialized := "Unit1.Em5.ControlNodes".em.status.initialized,
                      active := NOT (NOT "Unit1.Em5.ControlNodes".transferPnPLeft.selectJobStatus[2].active AND NOT "Unit1.Em5.ControlNodes".transferPnPLeft.selectJobStatus[3].active AND NOT "Unit1.Em5.ControlNodes".transferPnPLeft.selectJobStatus[4].active) OR NOT (NOT "Unit1.Em5.ControlNodes".transferPnPLeft.selectJobStatus[5].active AND NOT "Unit1.Em5.ControlNodes".transferPnPLeft.selectJobStatus[6].active AND NOT "Unit1.Em5.ControlNodes".transferPnPLeft.selectJobStatus[7].active) OR NOT (NOT "Unit1.Em5.ControlNodes".transferPnPLeft.selectJobStatus[9].active),
                      complete := "Unit1.Em5.ControlNodes".transferPnPLeft.sequence.status.stepComplete,
                      currentStep := "Unit1.Em5.ControlNodes".transferPnPLeft.sequence.status.currentStep,
                      stepCommand := "Unit1.Em5.ControlNodes".transferPnPLeft."step",
                      hmiStepStatus => "Unit1.Em5.HmiInterface".transferPnPLeft."step");
END_REGION

REGION Network 82: Call Transfer P&P Right Sequence
   RUNG wire#powerrail
      #InstSequenceTransferPnPRight(unitStatus := #statUnitStatus)
   END_RUNG
   // the same network as SCL:
   #InstSequenceTransferPnPRight(unitStatus := #statUnitStatus);   // "Unit1.Em5.Sequence_2_TransferPnPRight"
END_REGION

REGION Network 83: Transfer P&P Right
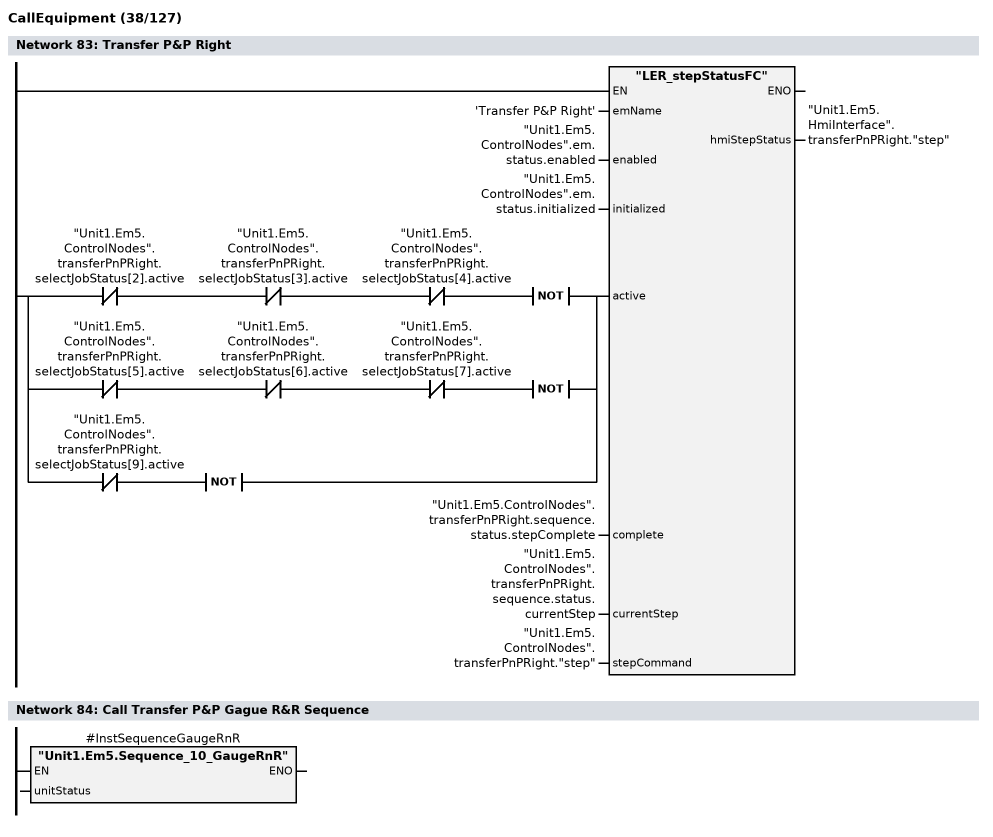
   RUNG wire#powerrail
      "LER_stepStatusFC"(active := wire#w1, emName := 'Transfer P&P Right', enabled := "Unit1.Em5.ControlNodes".em.status.enabled, initialized := "Unit1.Em5.ControlNodes".em.status.initialized, complete := "Unit1.Em5.ControlNodes".transferPnPRight.sequence.status.stepComplete, currentStep := "Unit1.Em5.ControlNodes".transferPnPRight.sequence.status.currentStep, stepCommand := "Unit1.Em5.ControlNodes".transferPnPRight."step", hmiStepStatus => "Unit1.Em5.HmiInterface".transferPnPRight."step")
   END_RUNG
   RUNG wire#powerrail
      I_Contact( "Unit1.Em5.ControlNodes".transferPnPRight.selectJobStatus[2].active )
      I_Contact( "Unit1.Em5.ControlNodes".transferPnPRight.selectJobStatus[3].active )
      I_Contact( "Unit1.Em5.ControlNodes".transferPnPRight.selectJobStatus[4].active )
      Not()
   END_RUNG wire#w1
   RUNG wire#powerrail
      I_Contact( "Unit1.Em5.ControlNodes".transferPnPRight.selectJobStatus[5].active )
      I_Contact( "Unit1.Em5.ControlNodes".transferPnPRight.selectJobStatus[6].active )
      I_Contact( "Unit1.Em5.ControlNodes".transferPnPRight.selectJobStatus[7].active )
      Not()
   END_RUNG wire#w1
   RUNG wire#powerrail
      I_Contact( "Unit1.Em5.ControlNodes".transferPnPRight.selectJobStatus[9].active )
      Not()
   END_RUNG wire#w1
   // the same network as SCL:
   "LER_stepStatusFC"(emName := 'Transfer P&P Right',
                      enabled := "Unit1.Em5.ControlNodes".em.status.enabled,
                      initialized := "Unit1.Em5.ControlNodes".em.status.initialized,
                      active := NOT (NOT "Unit1.Em5.ControlNodes".transferPnPRight.selectJobStatus[2].active AND NOT "Unit1.Em5.ControlNodes".transferPnPRight.selectJobStatus[3].active AND NOT "Unit1.Em5.ControlNodes".transferPnPRight.selectJobStatus[4].active) OR NOT (NOT "Unit1.Em5.ControlNodes".transferPnPRight.selectJobStatus[5].active AND NOT "Unit1.Em5.ControlNodes".transferPnPRight.selectJobStatus[6].active AND NOT "Unit1.Em5.ControlNodes".transferPnPRight.selectJobStatus[7].active) OR NOT (NOT "Unit1.Em5.ControlNodes".transferPnPRight.selectJobStatus[9].active),
                      complete := "Unit1.Em5.ControlNodes".transferPnPRight.sequence.status.stepComplete,
                      currentStep := "Unit1.Em5.ControlNodes".transferPnPRight.sequence.status.currentStep,
                      stepCommand := "Unit1.Em5.ControlNodes".transferPnPRight."step",
                      hmiStepStatus => "Unit1.Em5.HmiInterface".transferPnPRight."step");
END_REGION

REGION Network 84: Call Transfer P&P Gague R&R Sequence
   RUNG wire#powerrail
      #InstSequenceGaugeRnR(unitStatus :=)
   END_RUNG
   // the same network as SCL:
   #InstSequenceGaugeRnR();   // "Unit1.Em5.Sequence_10_GaugeRnR"
END_REGION

REGION Network 85: Transfer P&P Gague R&R Status
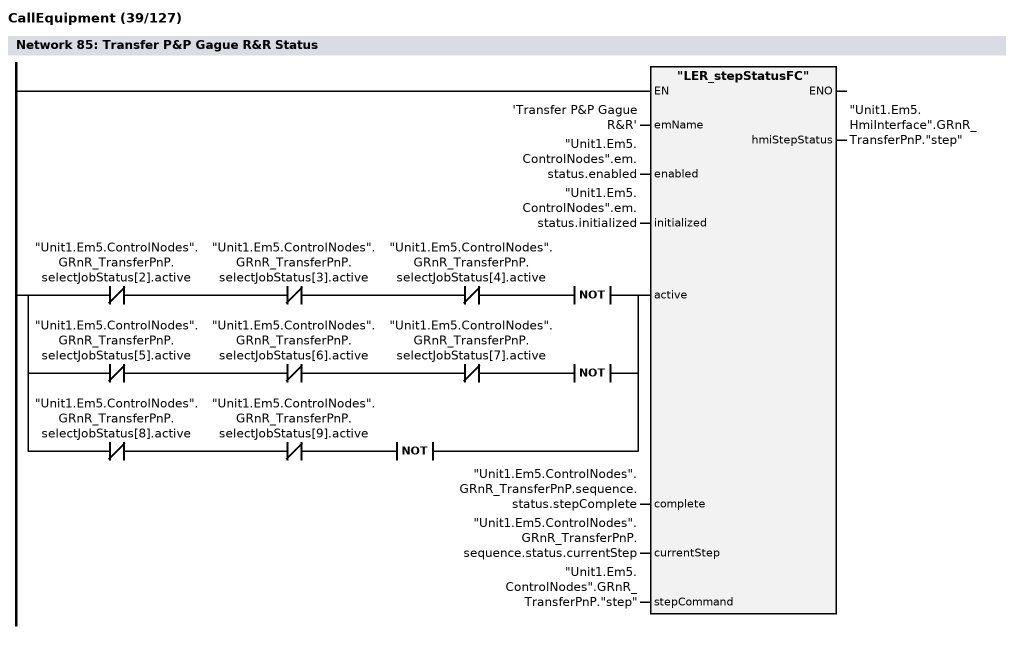
   RUNG wire#powerrail
      "LER_stepStatusFC"(active := wire#w1, emName := 'Transfer P&P Gague R&R', enabled := "Unit1.Em5.ControlNodes".em.status.enabled, initialized := "Unit1.Em5.ControlNodes".em.status.initialized, complete := "Unit1.Em5.ControlNodes".GRnR_TransferPnP.sequence.status.stepComplete, currentStep := "Unit1.Em5.ControlNodes".GRnR_TransferPnP.sequence.status.currentStep, stepCommand := "Unit1.Em5.ControlNodes".GRnR_TransferPnP."step", hmiStepStatus => "Unit1.Em5.HmiInterface".GRnR_TransferPnP."step")
   END_RUNG
   RUNG wire#powerrail
      I_Contact( "Unit1.Em5.ControlNodes".GRnR_TransferPnP.selectJobStatus[2].active )
      I_Contact( "Unit1.Em5.ControlNodes".GRnR_TransferPnP.selectJobStatus[3].active )
      I_Contact( "Unit1.Em5.ControlNodes".GRnR_TransferPnP.selectJobStatus[4].active )
      Not()
   END_RUNG wire#w1
   RUNG wire#powerrail
      I_Contact( "Unit1.Em5.ControlNodes".GRnR_TransferPnP.selectJobStatus[5].active )
      I_Contact( "Unit1.Em5.ControlNodes".GRnR_TransferPnP.selectJobStatus[6].active )
      I_Contact( "Unit1.Em5.ControlNodes".GRnR_TransferPnP.selectJobStatus[7].active )
      Not()
   END_RUNG wire#w1
   RUNG wire#powerrail
      I_Contact( "Unit1.Em5.ControlNodes".GRnR_TransferPnP.selectJobStatus[8].active )
      I_Contact( "Unit1.Em5.ControlNodes".GRnR_TransferPnP.selectJobStatus[9].active )
      Not()
   END_RUNG wire#w1
   // the same network as SCL:
   "LER_stepStatusFC"(emName := 'Transfer P&P Gague R&R',
                      enabled := "Unit1.Em5.ControlNodes".em.status.enabled,
                      initialized := "Unit1.Em5.ControlNodes".em.status.initialized,
                      active := NOT (NOT "Unit1.Em5.ControlNodes".GRnR_TransferPnP.selectJobStatus[2].active AND NOT "Unit1.Em5.ControlNodes".GRnR_TransferPnP.selectJobStatus[3].active AND NOT "Unit1.Em5.ControlNodes".GRnR_TransferPnP.selectJobStatus[4].active) OR NOT (NOT "Unit1.Em5.ControlNodes".GRnR_TransferPnP.selectJobStatus[5].active AND NOT "Unit1.Em5.ControlNodes".GRnR_TransferPnP.selectJobStatus[6].active AND NOT "Unit1.Em5.ControlNodes".GRnR_TransferPnP.selectJobStatus[7].active) OR NOT (NOT "Unit1.Em5.ControlNodes".GRnR_TransferPnP.selectJobStatus[8].active AND NOT "Unit1.Em5.ControlNodes".GRnR_TransferPnP.selectJobStatus[9].active),
                      complete := "Unit1.Em5.ControlNodes".GRnR_TransferPnP.sequence.status.stepComplete,
                      currentStep := "Unit1.Em5.ControlNodes".GRnR_TransferPnP.sequence.status.currentStep,
                      stepCommand := "Unit1.Em5.ControlNodes".GRnR_TransferPnP."step",
                      hmiStepStatus => "Unit1.Em5.HmiInterface".GRnR_TransferPnP."step");
END_REGION

REGION Network 87: ******************** Control Modules (Axis) ********************
   // Call control modules that are actuators after the em logic (jobs and sequence), so that the latest commands are applied to the actuators.
END_REGION

REGION Network 88: Reset CMS
   // Reset Axis when the unit is in the resetting state.
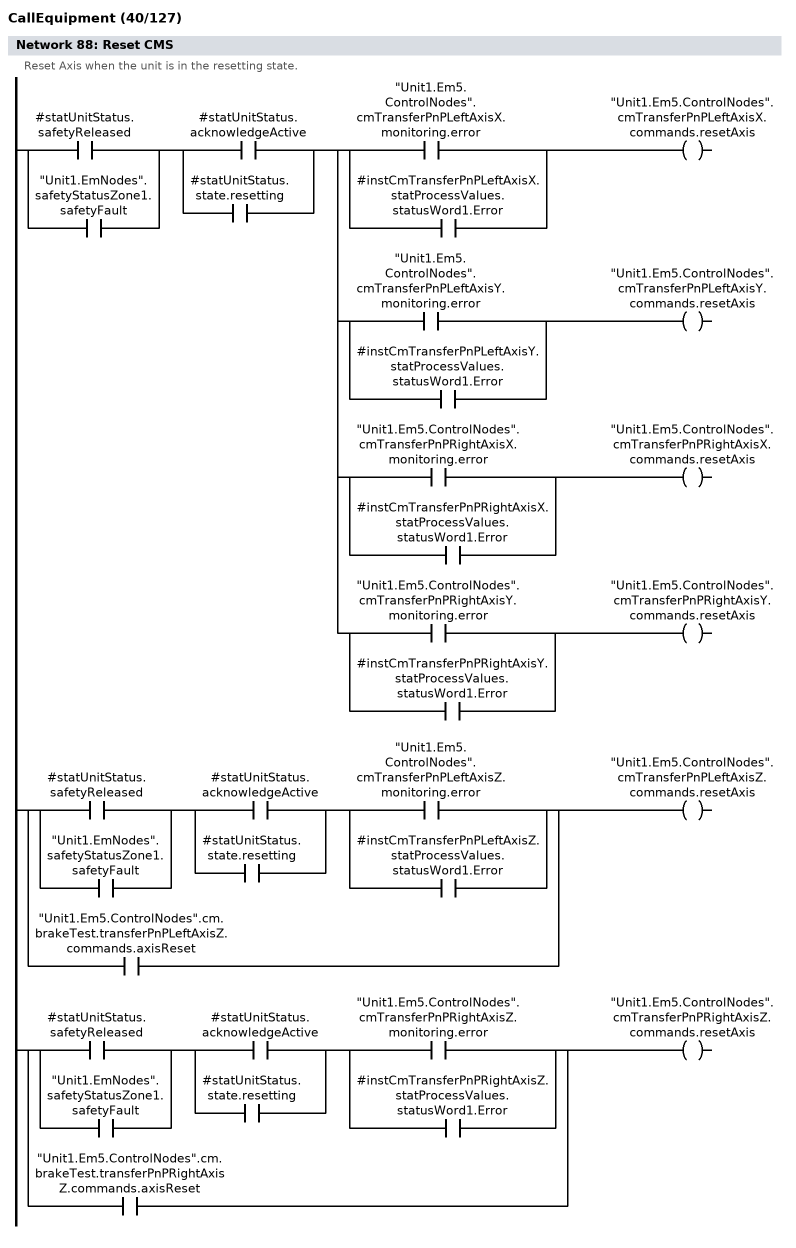
   RUNG wire#powerrail
      Contact( #statUnitStatus.safetyReleased )
      wire#w1
      Contact( #statUnitStatus.acknowledgeActive )
      wire#w2
      Contact( "Unit1.Em5.ControlNodes".cmTransferPnPLeftAxisX.monitoring.error )
      wire#w3
      Coil( "Unit1.Em5.ControlNodes".cmTransferPnPLeftAxisX.commands.resetAxis )
   END_RUNG
   RUNG wire#powerrail
      Contact( "Unit1.EmNodes".safetyStatusZone1.safetyFault )
   END_RUNG wire#w1
   RUNG wire#w1
      Contact( #statUnitStatus.state.resetting )
   END_RUNG wire#w2
   RUNG wire#w2
      Contact( #instCmTransferPnPLeftAxisX.statProcessValues.statusWord1.Error )
   END_RUNG wire#w3
   RUNG wire#w2
      Contact( "Unit1.Em5.ControlNodes".cmTransferPnPLeftAxisY.monitoring.error )
      wire#w4
      Coil( "Unit1.Em5.ControlNodes".cmTransferPnPLeftAxisY.commands.resetAxis )
   END_RUNG
   RUNG wire#w2
      Contact( #instCmTransferPnPLeftAxisY.statProcessValues.statusWord1.Error )
   END_RUNG wire#w4
   RUNG wire#w2
      Contact( "Unit1.Em5.ControlNodes".cmTransferPnPRightAxisX.monitoring.error )
      wire#w5
      Coil( "Unit1.Em5.ControlNodes".cmTransferPnPRightAxisX.commands.resetAxis )
   END_RUNG
   RUNG wire#w2
      Contact( #instCmTransferPnPRightAxisX.statProcessValues.statusWord1.Error )
   END_RUNG wire#w5
   RUNG wire#w2
      Contact( "Unit1.Em5.ControlNodes".cmTransferPnPRightAxisY.monitoring.error )
      wire#w6
      Coil( "Unit1.Em5.ControlNodes".cmTransferPnPRightAxisY.commands.resetAxis )
   END_RUNG
   RUNG wire#w2
      Contact( #instCmTransferPnPRightAxisY.statProcessValues.statusWord1.Error )
   END_RUNG wire#w6
   RUNG wire#powerrail
      Contact( #statUnitStatus.safetyReleased )
      wire#w7
      Contact( #statUnitStatus.acknowledgeActive )
      wire#w8
      Contact( "Unit1.Em5.ControlNodes".cmTransferPnPLeftAxisZ.monitoring.error )
      wire#w9
      Coil( "Unit1.Em5.ControlNodes".cmTransferPnPLeftAxisZ.commands.resetAxis )
   END_RUNG
   RUNG wire#powerrail
      Contact( "Unit1.EmNodes".safetyStatusZone1.safetyFault )
   END_RUNG wire#w7
   RUNG wire#w7
      Contact( #statUnitStatus.state.resetting )
   END_RUNG wire#w8
   RUNG wire#w8
      Contact( #instCmTransferPnPLeftAxisZ.statProcessValues.statusWord1.Error )
   END_RUNG wire#w9
   RUNG wire#powerrail
      Contact( "Unit1.Em5.ControlNodes".cm.brakeTest.transferPnPLeftAxisZ.commands.axisReset )
   END_RUNG wire#w9
   RUNG wire#powerrail
      Contact( #statUnitStatus.safetyReleased )
      wire#w10
      Contact( #statUnitStatus.acknowledgeActive )
      wire#w11
      Contact( "Unit1.Em5.ControlNodes".cmTransferPnPRightAxisZ.monitoring.error )
      wire#w12
      Coil( "Unit1.Em5.ControlNodes".cmTransferPnPRightAxisZ.commands.resetAxis )
   END_RUNG
   RUNG wire#powerrail
      Contact( "Unit1.EmNodes".safetyStatusZone1.safetyFault )
   END_RUNG wire#w10
   RUNG wire#w10
      Contact( #statUnitStatus.state.resetting )
   END_RUNG wire#w11
   RUNG wire#w11
      Contact( #instCmTransferPnPRightAxisZ.statProcessValues.statusWord1.Error )
   END_RUNG wire#w12
   RUNG wire#powerrail
      Contact( "Unit1.Em5.ControlNodes".cm.brakeTest.transferPnPRightAxisZ.commands.axisReset )
   END_RUNG wire#w12
   // the same network as SCL:
   #_w1 := (#statUnitStatus.safetyReleased OR "Unit1.EmNodes".safetyStatusZone1.safetyFault) AND (#statUnitStatus.acknowledgeActive OR #statUnitStatus.state.resetting);
   "Unit1.Em5.ControlNodes".cmTransferPnPLeftAxisX.commands.resetAxis := #_w1 AND ("Unit1.Em5.ControlNodes".cmTransferPnPLeftAxisX.monitoring.error OR #instCmTransferPnPLeftAxisX.statProcessValues.statusWord1.Error);
   "Unit1.Em5.ControlNodes".cmTransferPnPLeftAxisY.commands.resetAxis := #_w1 AND ("Unit1.Em5.ControlNodes".cmTransferPnPLeftAxisY.monitoring.error OR #instCmTransferPnPLeftAxisY.statProcessValues.statusWord1.Error);
   "Unit1.Em5.ControlNodes".cmTransferPnPRightAxisX.commands.resetAxis := #_w1 AND ("Unit1.Em5.ControlNodes".cmTransferPnPRightAxisX.monitoring.error OR #instCmTransferPnPRightAxisX.statProcessValues.statusWord1.Error);
   "Unit1.Em5.ControlNodes".cmTransferPnPRightAxisY.commands.resetAxis := #_w1 AND ("Unit1.Em5.ControlNodes".cmTransferPnPRightAxisY.monitoring.error OR #instCmTransferPnPRightAxisY.statProcessValues.statusWord1.Error);
   "Unit1.Em5.ControlNodes".cmTransferPnPLeftAxisZ.commands.resetAxis := ((#statUnitStatus.safetyReleased OR "Unit1.EmNodes".safetyStatusZone1.safetyFault) AND (#statUnitStatus.acknowledgeActive OR #statUnitStatus.state.resetting) AND ("Unit1.Em5.ControlNodes".cmTransferPnPLeftAxisZ.monitoring.error OR #instCmTransferPnPLeftAxisZ.statProcessValues.statusWord1.Error)) OR "Unit1.Em5.ControlNodes".cm.brakeTest.transferPnPLeftAxisZ.commands.axisReset;
   "Unit1.Em5.ControlNodes".cmTransferPnPRightAxisZ.commands.resetAxis := ((#statUnitStatus.safetyReleased OR "Unit1.EmNodes".safetyStatusZone1.safetyFault) AND (#statUnitStatus.acknowledgeActive OR #statUnitStatus.state.resetting) AND ("Unit1.Em5.ControlNodes".cmTransferPnPRightAxisZ.monitoring.error OR #instCmTransferPnPRightAxisZ.statProcessValues.statusWord1.Error)) OR "Unit1.Em5.ControlNodes".cm.brakeTest.transferPnPRightAxisZ.commands.axisReset;
END_REGION

REGION Network 89: Enable/Disable CMs
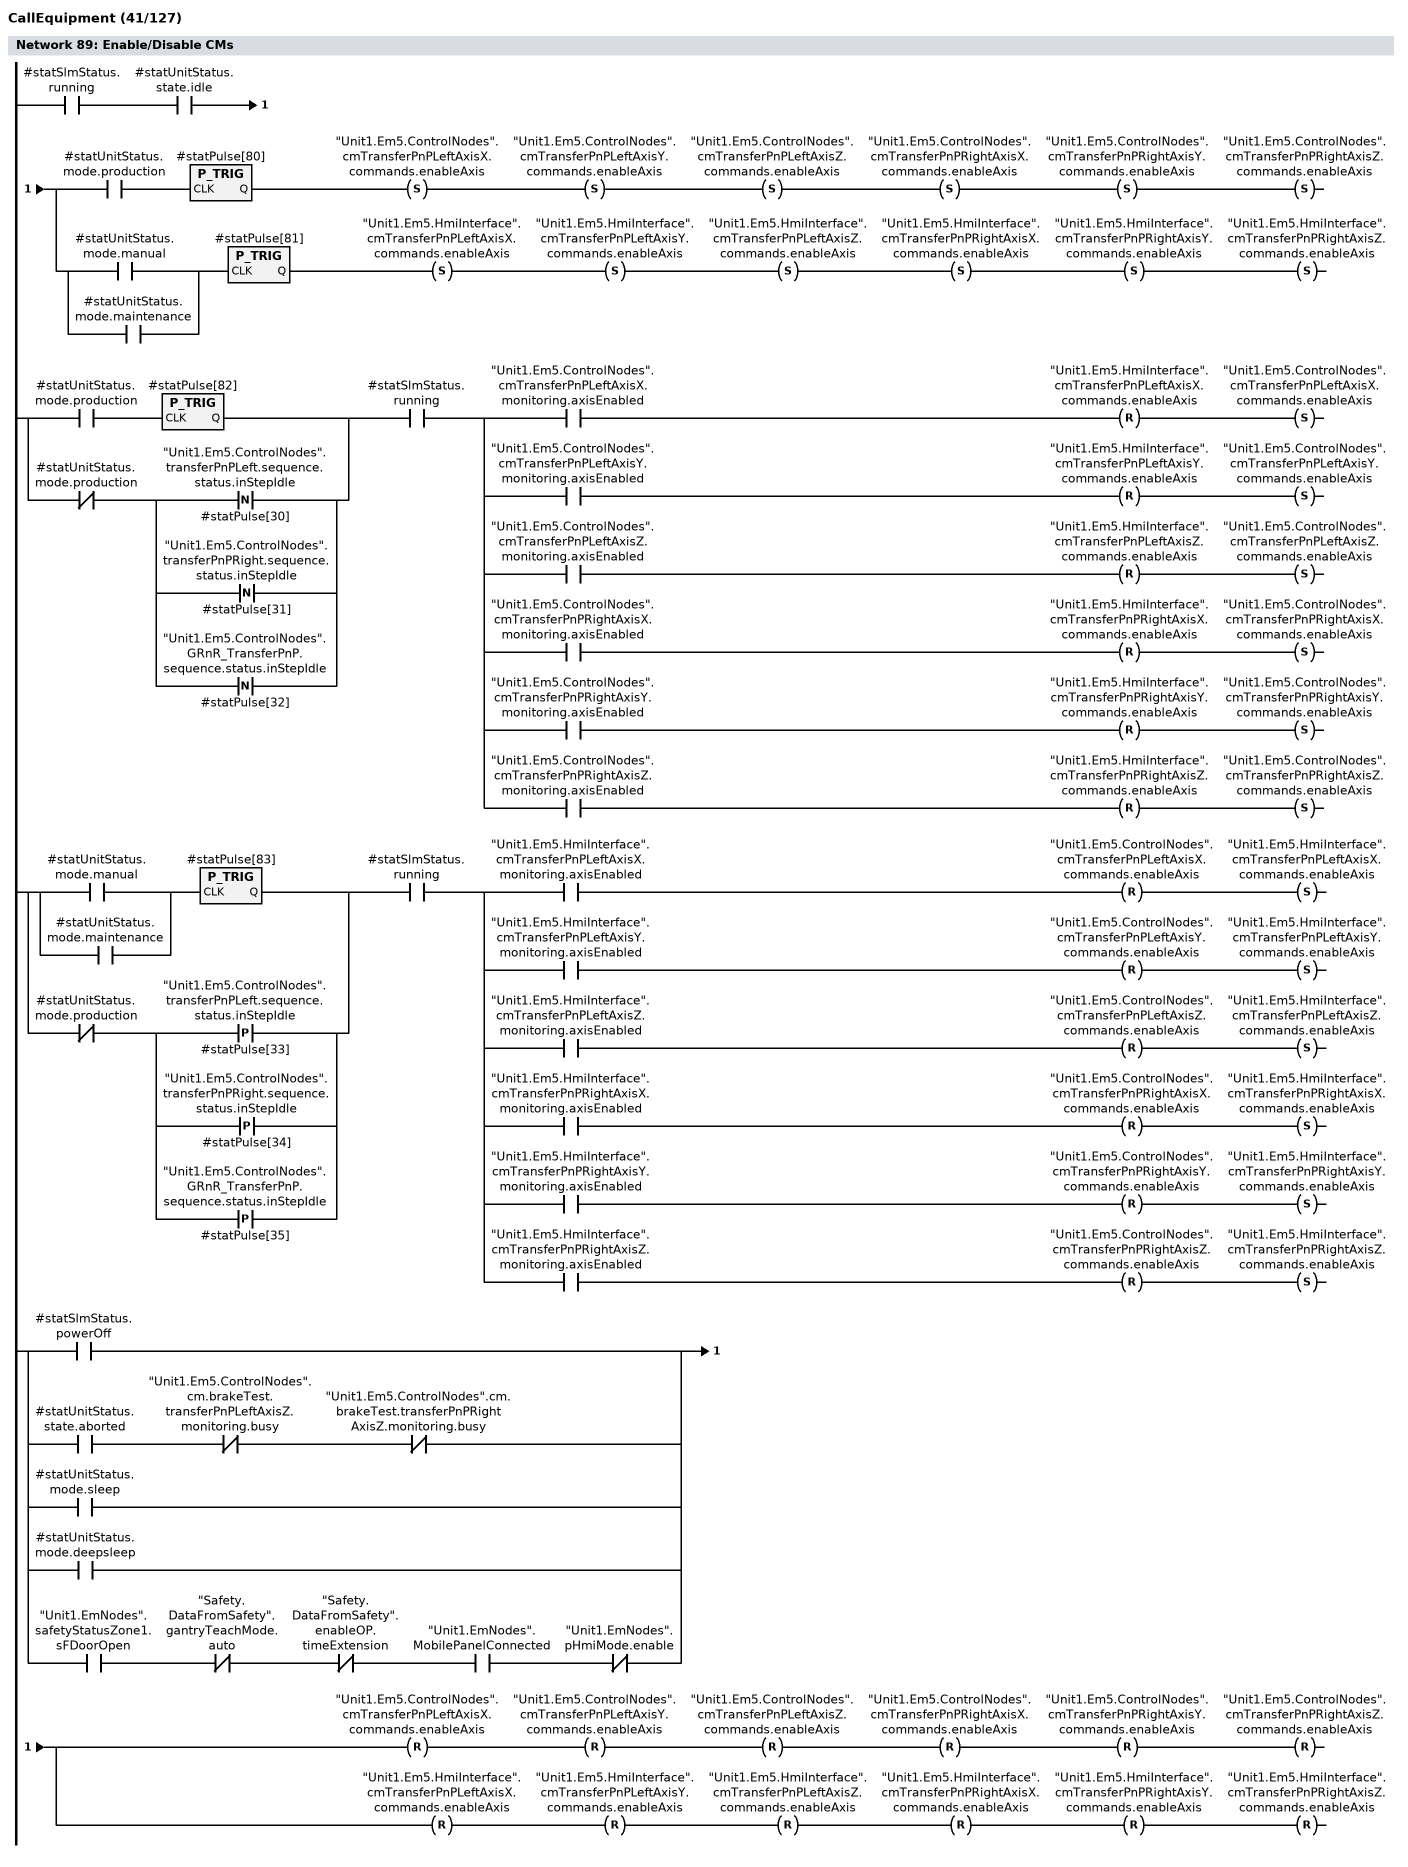
   RUNG wire#powerrail
      Contact( #statSlmStatus.running )
      Contact( #statUnitStatus.state.idle )
      wire#w1
      Contact( #statUnitStatus.mode.production )
      P_Trig( #statPulse[80] )
      S_Coil( "Unit1.Em5.ControlNodes".cmTransferPnPLeftAxisX.commands.enableAxis )
      S_Coil( "Unit1.Em5.ControlNodes".cmTransferPnPLeftAxisY.commands.enableAxis )
      S_Coil( "Unit1.Em5.ControlNodes".cmTransferPnPLeftAxisZ.commands.enableAxis )
      S_Coil( "Unit1.Em5.ControlNodes".cmTransferPnPRightAxisX.commands.enableAxis )
      S_Coil( "Unit1.Em5.ControlNodes".cmTransferPnPRightAxisY.commands.enableAxis )
      S_Coil( "Unit1.Em5.ControlNodes".cmTransferPnPRightAxisZ.commands.enableAxis )
   END_RUNG
   RUNG wire#w1
      Contact( #statUnitStatus.mode.manual )
      wire#w2
      P_Trig( #statPulse[81] )
      S_Coil( "Unit1.Em5.HmiInterface".cmTransferPnPLeftAxisX.commands.enableAxis )
      S_Coil( "Unit1.Em5.HmiInterface".cmTransferPnPLeftAxisY.commands.enableAxis )
      S_Coil( "Unit1.Em5.HmiInterface".cmTransferPnPLeftAxisZ.commands.enableAxis )
      S_Coil( "Unit1.Em5.HmiInterface".cmTransferPnPRightAxisX.commands.enableAxis )
      S_Coil( "Unit1.Em5.HmiInterface".cmTransferPnPRightAxisY.commands.enableAxis )
      S_Coil( "Unit1.Em5.HmiInterface".cmTransferPnPRightAxisZ.commands.enableAxis )
   END_RUNG
   RUNG wire#w1
      Contact( #statUnitStatus.mode.maintenance )
   END_RUNG wire#w2
   RUNG wire#powerrail
      Contact( #statUnitStatus.mode.production )
      P_Trig( #statPulse[82] )
      wire#w3
      Contact( #statSlmStatus.running )
      wire#w5
      Contact( "Unit1.Em5.ControlNodes".cmTransferPnPLeftAxisX.monitoring.axisEnabled )
      R_Coil( "Unit1.Em5.HmiInterface".cmTransferPnPLeftAxisX.commands.enableAxis )
      S_Coil( "Unit1.Em5.ControlNodes".cmTransferPnPLeftAxisX.commands.enableAxis )
   END_RUNG
   RUNG wire#powerrail
      I_Contact( #statUnitStatus.mode.production )
      wire#w4
      N_Contact(operand := "Unit1.Em5.ControlNodes".transferPnPLeft.sequence.status.inStepIdle, bit := #statPulse[30])
   END_RUNG wire#w3
   RUNG wire#w4
      N_Contact(operand := "Unit1.Em5.ControlNodes".transferPnPRight.sequence.status.inStepIdle, bit := #statPulse[31])
   END_RUNG wire#w3
   RUNG wire#w4
      N_Contact(operand := "Unit1.Em5.ControlNodes".GRnR_TransferPnP.sequence.status.inStepIdle, bit := #statPulse[32])
   END_RUNG wire#w3
   RUNG wire#w5
      Contact( "Unit1.Em5.ControlNodes".cmTransferPnPLeftAxisY.monitoring.axisEnabled )
      R_Coil( "Unit1.Em5.HmiInterface".cmTransferPnPLeftAxisY.commands.enableAxis )
      S_Coil( "Unit1.Em5.ControlNodes".cmTransferPnPLeftAxisY.commands.enableAxis )
   END_RUNG
   RUNG wire#w5
      Contact( "Unit1.Em5.ControlNodes".cmTransferPnPLeftAxisZ.monitoring.axisEnabled )
      R_Coil( "Unit1.Em5.HmiInterface".cmTransferPnPLeftAxisZ.commands.enableAxis )
      S_Coil( "Unit1.Em5.ControlNodes".cmTransferPnPLeftAxisZ.commands.enableAxis )
   END_RUNG
   RUNG wire#w5
      Contact( "Unit1.Em5.ControlNodes".cmTransferPnPRightAxisX.monitoring.axisEnabled )
      R_Coil( "Unit1.Em5.HmiInterface".cmTransferPnPRightAxisX.commands.enableAxis )
      S_Coil( "Unit1.Em5.ControlNodes".cmTransferPnPRightAxisX.commands.enableAxis )
   END_RUNG
   RUNG wire#w5
      Contact( "Unit1.Em5.ControlNodes".cmTransferPnPRightAxisY.monitoring.axisEnabled )
      R_Coil( "Unit1.Em5.HmiInterface".cmTransferPnPRightAxisY.commands.enableAxis )
      S_Coil( "Unit1.Em5.ControlNodes".cmTransferPnPRightAxisY.commands.enableAxis )
   END_RUNG
   RUNG wire#w5
      Contact( "Unit1.Em5.ControlNodes".cmTransferPnPRightAxisZ.monitoring.axisEnabled )
      R_Coil( "Unit1.Em5.HmiInterface".cmTransferPnPRightAxisZ.commands.enableAxis )
      S_Coil( "Unit1.Em5.ControlNodes".cmTransferPnPRightAxisZ.commands.enableAxis )
   END_RUNG
   RUNG wire#powerrail
      Contact( #statUnitStatus.mode.manual )
      wire#w6
      P_Trig( #statPulse[83] )
      wire#w7
      Contact( #statSlmStatus.running )
      wire#w9
      Contact( "Unit1.Em5.HmiInterface".cmTransferPnPLeftAxisX.monitoring.axisEnabled )
      R_Coil( "Unit1.Em5.ControlNodes".cmTransferPnPLeftAxisX.commands.enableAxis )
      S_Coil( "Unit1.Em5.HmiInterface".cmTransferPnPLeftAxisX.commands.enableAxis )
   END_RUNG
   RUNG wire#powerrail
      Contact( #statUnitStatus.mode.maintenance )
   END_RUNG wire#w6
   RUNG wire#powerrail
      I_Contact( #statUnitStatus.mode.production )
      wire#w8
      P_Contact(operand := "Unit1.Em5.ControlNodes".transferPnPLeft.sequence.status.inStepIdle, bit := #statPulse[33])
   END_RUNG wire#w7
   RUNG wire#w8
      P_Contact(operand := "Unit1.Em5.ControlNodes".transferPnPRight.sequence.status.inStepIdle, bit := #statPulse[34])
   END_RUNG wire#w7
   RUNG wire#w8
      P_Contact(operand := "Unit1.Em5.ControlNodes".GRnR_TransferPnP.sequence.status.inStepIdle, bit := #statPulse[35])
   END_RUNG wire#w7
   RUNG wire#w9
      Contact( "Unit1.Em5.HmiInterface".cmTransferPnPLeftAxisY.monitoring.axisEnabled )
      R_Coil( "Unit1.Em5.ControlNodes".cmTransferPnPLeftAxisY.commands.enableAxis )
      S_Coil( "Unit1.Em5.HmiInterface".cmTransferPnPLeftAxisY.commands.enableAxis )
   END_RUNG
   RUNG wire#w9
      Contact( "Unit1.Em5.HmiInterface".cmTransferPnPLeftAxisZ.monitoring.axisEnabled )
      R_Coil( "Unit1.Em5.ControlNodes".cmTransferPnPLeftAxisZ.commands.enableAxis )
      S_Coil( "Unit1.Em5.HmiInterface".cmTransferPnPLeftAxisZ.commands.enableAxis )
   END_RUNG
   RUNG wire#w9
      Contact( "Unit1.Em5.HmiInterface".cmTransferPnPRightAxisX.monitoring.axisEnabled )
      R_Coil( "Unit1.Em5.ControlNodes".cmTransferPnPRightAxisX.commands.enableAxis )
      S_Coil( "Unit1.Em5.HmiInterface".cmTransferPnPRightAxisX.commands.enableAxis )
   END_RUNG
   RUNG wire#w9
      Contact( "Unit1.Em5.HmiInterface".cmTransferPnPRightAxisY.monitoring.axisEnabled )
      R_Coil( "Unit1.Em5.ControlNodes".cmTransferPnPRightAxisY.commands.enableAxis )
      S_Coil( "Unit1.Em5.HmiInterface".cmTransferPnPRightAxisY.commands.enableAxis )
   END_RUNG
   RUNG wire#w9
      Contact( "Unit1.Em5.HmiInterface".cmTransferPnPRightAxisZ.monitoring.axisEnabled )
      R_Coil( "Unit1.Em5.ControlNodes".cmTransferPnPRightAxisZ.commands.enableAxis )
      S_Coil( "Unit1.Em5.HmiInterface".cmTransferPnPRightAxisZ.commands.enableAxis )
   END_RUNG
   RUNG wire#powerrail
      Contact( #statSlmStatus.powerOff )
      wire#w10
      R_Coil( "Unit1.Em5.ControlNodes".cmTransferPnPLeftAxisX.commands.enableAxis )
      R_Coil( "Unit1.Em5.ControlNodes".cmTransferPnPLeftAxisY.commands.enableAxis )
      R_Coil( "Unit1.Em5.ControlNodes".cmTransferPnPLeftAxisZ.commands.enableAxis )
      R_Coil( "Unit1.Em5.ControlNodes".cmTransferPnPRightAxisX.commands.enableAxis )
      R_Coil( "Unit1.Em5.ControlNodes".cmTransferPnPRightAxisY.commands.enableAxis )
      R_Coil( "Unit1.Em5.ControlNodes".cmTransferPnPRightAxisZ.commands.enableAxis )
   END_RUNG
   RUNG wire#powerrail
      Contact( #statUnitStatus.state.aborted )
      I_Contact( "Unit1.Em5.ControlNodes".cm.brakeTest.transferPnPLeftAxisZ.monitoring.busy )
      I_Contact( "Unit1.Em5.ControlNodes".cm.brakeTest.transferPnPRightAxisZ.monitoring.busy )
   END_RUNG wire#w10
   RUNG wire#powerrail
      Contact( #statUnitStatus.mode.sleep )
   END_RUNG wire#w10
   RUNG wire#powerrail
      Contact( #statUnitStatus.mode.deepsleep )
   END_RUNG wire#w10
   RUNG wire#powerrail
      Contact( "Unit1.EmNodes".safetyStatusZone1.sFDoorOpen )
      I_Contact( "Safety.DataFromSafety".gantryTeachMode.auto )
      I_Contact( "Safety.DataFromSafety".enableOP.timeExtension )
      Contact( "Unit1.EmNodes".MobilePanelConnected )
      I_Contact( "Unit1.EmNodes".pHmiMode.enable )
   END_RUNG wire#w10
   RUNG wire#w10
      R_Coil( "Unit1.Em5.HmiInterface".cmTransferPnPLeftAxisX.commands.enableAxis )
      R_Coil( "Unit1.Em5.HmiInterface".cmTransferPnPLeftAxisY.commands.enableAxis )
      R_Coil( "Unit1.Em5.HmiInterface".cmTransferPnPLeftAxisZ.commands.enableAxis )
      R_Coil( "Unit1.Em5.HmiInterface".cmTransferPnPRightAxisX.commands.enableAxis )
      R_Coil( "Unit1.Em5.HmiInterface".cmTransferPnPRightAxisY.commands.enableAxis )
      R_Coil( "Unit1.Em5.HmiInterface".cmTransferPnPRightAxisZ.commands.enableAxis )
   END_RUNG
   // the same network as SCL:
   #_w1 := #statSlmStatus.running AND #statUnitStatus.state.idle;
   #_w2 := #_w1 AND #statUnitStatus.mode.production;
   #_w3 := #_w2 AND NOT #statPulse[80];   // rising edge
   #statPulse[80] := #_w2;
   IF #_w3 THEN
       "Unit1.Em5.ControlNodes".cmTransferPnPLeftAxisX.commands.enableAxis := TRUE;
       "Unit1.Em5.ControlNodes".cmTransferPnPLeftAxisY.commands.enableAxis := TRUE;
       "Unit1.Em5.ControlNodes".cmTransferPnPLeftAxisZ.commands.enableAxis := TRUE;
       "Unit1.Em5.ControlNodes".cmTransferPnPRightAxisX.commands.enableAxis := TRUE;
       "Unit1.Em5.ControlNodes".cmTransferPnPRightAxisY.commands.enableAxis := TRUE;
       "Unit1.Em5.ControlNodes".cmTransferPnPRightAxisZ.commands.enableAxis := TRUE;
   END_IF;
   #_w4 := #_w1 AND (#statUnitStatus.mode.manual OR #statUnitStatus.mode.maintenance);
   #_w5 := #_w4 AND NOT #statPulse[81];   // rising edge
   #statPulse[81] := #_w4;
   IF #_w5 THEN
       "Unit1.Em5.HmiInterface".cmTransferPnPLeftAxisX.commands.enableAxis := TRUE;
       "Unit1.Em5.HmiInterface".cmTransferPnPLeftAxisY.commands.enableAxis := TRUE;
       "Unit1.Em5.HmiInterface".cmTransferPnPLeftAxisZ.commands.enableAxis := TRUE;
       "Unit1.Em5.HmiInterface".cmTransferPnPRightAxisX.commands.enableAxis := TRUE;
       "Unit1.Em5.HmiInterface".cmTransferPnPRightAxisY.commands.enableAxis := TRUE;
       "Unit1.Em5.HmiInterface".cmTransferPnPRightAxisZ.commands.enableAxis := TRUE;
   END_IF;
   #_w6 := #statUnitStatus.mode.production AND NOT #statPulse[82];   // rising edge
   #statPulse[82] := #statUnitStatus.mode.production;
   #_w7 := NOT #statUnitStatus.mode.production AND NOT "Unit1.Em5.ControlNodes".transferPnPLeft.sequence.status.inStepIdle AND #statPulse[30];   // falling edge of "Unit1.Em5.ControlNodes".transferPnPLeft.sequence.status.inStepIdle
   #statPulse[30] := "Unit1.Em5.ControlNodes".transferPnPLeft.sequence.status.inStepIdle;
   #_w8 := NOT #statUnitStatus.mode.production AND NOT "Unit1.Em5.ControlNodes".transferPnPRight.sequence.status.inStepIdle AND #statPulse[31];   // falling edge of "Unit1.Em5.ControlNodes".transferPnPRight.sequence.status.inStepIdle
   #statPulse[31] := "Unit1.Em5.ControlNodes".transferPnPRight.sequence.status.inStepIdle;
   #_w9 := NOT #statUnitStatus.mode.production AND NOT "Unit1.Em5.ControlNodes".GRnR_TransferPnP.sequence.status.inStepIdle AND #statPulse[32];   // falling edge of "Unit1.Em5.ControlNodes".GRnR_TransferPnP.sequence.status.inStepIdle
   #statPulse[32] := "Unit1.Em5.ControlNodes".GRnR_TransferPnP.sequence.status.inStepIdle;
   #_w10 := (#_w6 OR #_w7 OR #_w8 OR #_w9) AND #statSlmStatus.running;
   IF #_w10 AND "Unit1.Em5.ControlNodes".cmTransferPnPLeftAxisX.monitoring.axisEnabled THEN
       "Unit1.Em5.HmiInterface".cmTransferPnPLeftAxisX.commands.enableAxis := FALSE;
       "Unit1.Em5.ControlNodes".cmTransferPnPLeftAxisX.commands.enableAxis := TRUE;
   END_IF;
   IF #_w10 AND "Unit1.Em5.ControlNodes".cmTransferPnPLeftAxisY.monitoring.axisEnabled THEN
       "Unit1.Em5.HmiInterface".cmTransferPnPLeftAxisY.commands.enableAxis := FALSE;
       "Unit1.Em5.ControlNodes".cmTransferPnPLeftAxisY.commands.enableAxis := TRUE;
   END_IF;
   IF #_w10 AND "Unit1.Em5.ControlNodes".cmTransferPnPLeftAxisZ.monitoring.axisEnabled THEN
       "Unit1.Em5.HmiInterface".cmTransferPnPLeftAxisZ.commands.enableAxis := FALSE;
       "Unit1.Em5.ControlNodes".cmTransferPnPLeftAxisZ.commands.enableAxis := TRUE;
   END_IF;
   IF #_w10 AND "Unit1.Em5.ControlNodes".cmTransferPnPRightAxisX.monitoring.axisEnabled THEN
       "Unit1.Em5.HmiInterface".cmTransferPnPRightAxisX.commands.enableAxis := FALSE;
       "Unit1.Em5.ControlNodes".cmTransferPnPRightAxisX.commands.enableAxis := TRUE;
   END_IF;
   IF #_w10 AND "Unit1.Em5.ControlNodes".cmTransferPnPRightAxisY.monitoring.axisEnabled THEN
       "Unit1.Em5.HmiInterface".cmTransferPnPRightAxisY.commands.enableAxis := FALSE;
       "Unit1.Em5.ControlNodes".cmTransferPnPRightAxisY.commands.enableAxis := TRUE;
   END_IF;
   IF #_w10 AND "Unit1.Em5.ControlNodes".cmTransferPnPRightAxisZ.monitoring.axisEnabled THEN
       "Unit1.Em5.HmiInterface".cmTransferPnPRightAxisZ.commands.enableAxis := FALSE;
       "Unit1.Em5.ControlNodes".cmTransferPnPRightAxisZ.commands.enableAxis := TRUE;
   END_IF;
   #_w11 := #statUnitStatus.mode.manual OR #statUnitStatus.mode.maintenance;
   #_w12 := #_w11 AND NOT #statPulse[83];   // rising edge
   #statPulse[83] := #_w11;
   #_w13 := NOT #statUnitStatus.mode.production AND "Unit1.Em5.ControlNodes".transferPnPLeft.sequence.status.inStepIdle AND NOT #statPulse[33];   // rising edge of "Unit1.Em5.ControlNodes".transferPnPLeft.sequence.status.inStepIdle
   #statPulse[33] := "Unit1.Em5.ControlNodes".transferPnPLeft.sequence.status.inStepIdle;
   #_w14 := NOT #statUnitStatus.mode.production AND "Unit1.Em5.ControlNodes".transferPnPRight.sequence.status.inStepIdle AND NOT #statPulse[34];   // rising edge of "Unit1.Em5.ControlNodes".transferPnPRight.sequence.status.inStepIdle
   #statPulse[34] := "Unit1.Em5.ControlNodes".transferPnPRight.sequence.status.inStepIdle;
   #_w15 := NOT #statUnitStatus.mode.production AND "Unit1.Em5.ControlNodes".GRnR_TransferPnP.sequence.status.inStepIdle AND NOT #statPulse[35];   // rising edge of "Unit1.Em5.ControlNodes".GRnR_TransferPnP.sequence.status.inStepIdle
   #statPulse[35] := "Unit1.Em5.ControlNodes".GRnR_TransferPnP.sequence.status.inStepIdle;
   #_w16 := (#_w12 OR #_w13 OR #_w14 OR #_w15) AND #statSlmStatus.running;
   IF #_w16 AND "Unit1.Em5.HmiInterface".cmTransferPnPLeftAxisX.monitoring.axisEnabled THEN
       "Unit1.Em5.ControlNodes".cmTransferPnPLeftAxisX.commands.enableAxis := FALSE;
       "Unit1.Em5.HmiInterface".cmTransferPnPLeftAxisX.commands.enableAxis := TRUE;
   END_IF;
   IF #_w16 AND "Unit1.Em5.HmiInterface".cmTransferPnPLeftAxisY.monitoring.axisEnabled THEN
       "Unit1.Em5.ControlNodes".cmTransferPnPLeftAxisY.commands.enableAxis := FALSE;
       "Unit1.Em5.HmiInterface".cmTransferPnPLeftAxisY.commands.enableAxis := TRUE;
   END_IF;
   IF #_w16 AND "Unit1.Em5.HmiInterface".cmTransferPnPLeftAxisZ.monitoring.axisEnabled THEN
       "Unit1.Em5.ControlNodes".cmTransferPnPLeftAxisZ.commands.enableAxis := FALSE;
       "Unit1.Em5.HmiInterface".cmTransferPnPLeftAxisZ.commands.enableAxis := TRUE;
   END_IF;
   IF #_w16 AND "Unit1.Em5.HmiInterface".cmTransferPnPRightAxisX.monitoring.axisEnabled THEN
       "Unit1.Em5.ControlNodes".cmTransferPnPRightAxisX.commands.enableAxis := FALSE;
       "Unit1.Em5.HmiInterface".cmTransferPnPRightAxisX.commands.enableAxis := TRUE;
   END_IF;
   IF #_w16 AND "Unit1.Em5.HmiInterface".cmTransferPnPRightAxisY.monitoring.axisEnabled THEN
       "Unit1.Em5.ControlNodes".cmTransferPnPRightAxisY.commands.enableAxis := FALSE;
       "Unit1.Em5.HmiInterface".cmTransferPnPRightAxisY.commands.enableAxis := TRUE;
   END_IF;
   IF #_w16 AND "Unit1.Em5.HmiInterface".cmTransferPnPRightAxisZ.monitoring.axisEnabled THEN
       "Unit1.Em5.ControlNodes".cmTransferPnPRightAxisZ.commands.enableAxis := FALSE;
       "Unit1.Em5.HmiInterface".cmTransferPnPRightAxisZ.commands.enableAxis := TRUE;
   END_IF;
   IF #statSlmStatus.powerOff OR (#statUnitStatus.state.aborted AND NOT "Unit1.Em5.ControlNodes".cm.brakeTest.transferPnPLeftAxisZ.monitoring.busy AND NOT "Unit1.Em5.ControlNodes".cm.brakeTest.transferPnPRightAxisZ.monitoring.busy) OR #statUnitStatus.mode.sleep OR #statUnitStatus.mode.deepsleep OR ("Unit1.EmNodes".safetyStatusZone1.sFDoorOpen AND NOT "Safety.DataFromSafety".gantryTeachMode.auto AND NOT "Safety.DataFromSafety".enableOP.timeExtension AND "Unit1.EmNodes".MobilePanelConnected AND NOT "Unit1.EmNodes".pHmiMode.enable) THEN
       "Unit1.Em5.ControlNodes".cmTransferPnPLeftAxisX.commands.enableAxis := FALSE;
       "Unit1.Em5.ControlNodes".cmTransferPnPLeftAxisY.commands.enableAxis := FALSE;
       "Unit1.Em5.ControlNodes".cmTransferPnPLeftAxisZ.commands.enableAxis := FALSE;
       "Unit1.Em5.ControlNodes".cmTransferPnPRightAxisX.commands.enableAxis := FALSE;
       "Unit1.Em5.ControlNodes".cmTransferPnPRightAxisY.commands.enableAxis := FALSE;
       "Unit1.Em5.ControlNodes".cmTransferPnPRightAxisZ.commands.enableAxis := FALSE;
       "Unit1.Em5.HmiInterface".cmTransferPnPLeftAxisX.commands.enableAxis := FALSE;
       "Unit1.Em5.HmiInterface".cmTransferPnPLeftAxisY.commands.enableAxis := FALSE;
       "Unit1.Em5.HmiInterface".cmTransferPnPLeftAxisZ.commands.enableAxis := FALSE;
       "Unit1.Em5.HmiInterface".cmTransferPnPRightAxisX.commands.enableAxis := FALSE;
       "Unit1.Em5.HmiInterface".cmTransferPnPRightAxisY.commands.enableAxis := FALSE;
       "Unit1.Em5.HmiInterface".cmTransferPnPRightAxisZ.commands.enableAxis := FALSE;
   END_IF;
END_REGION

REGION Network 90: PHMI Servo Enable CMs
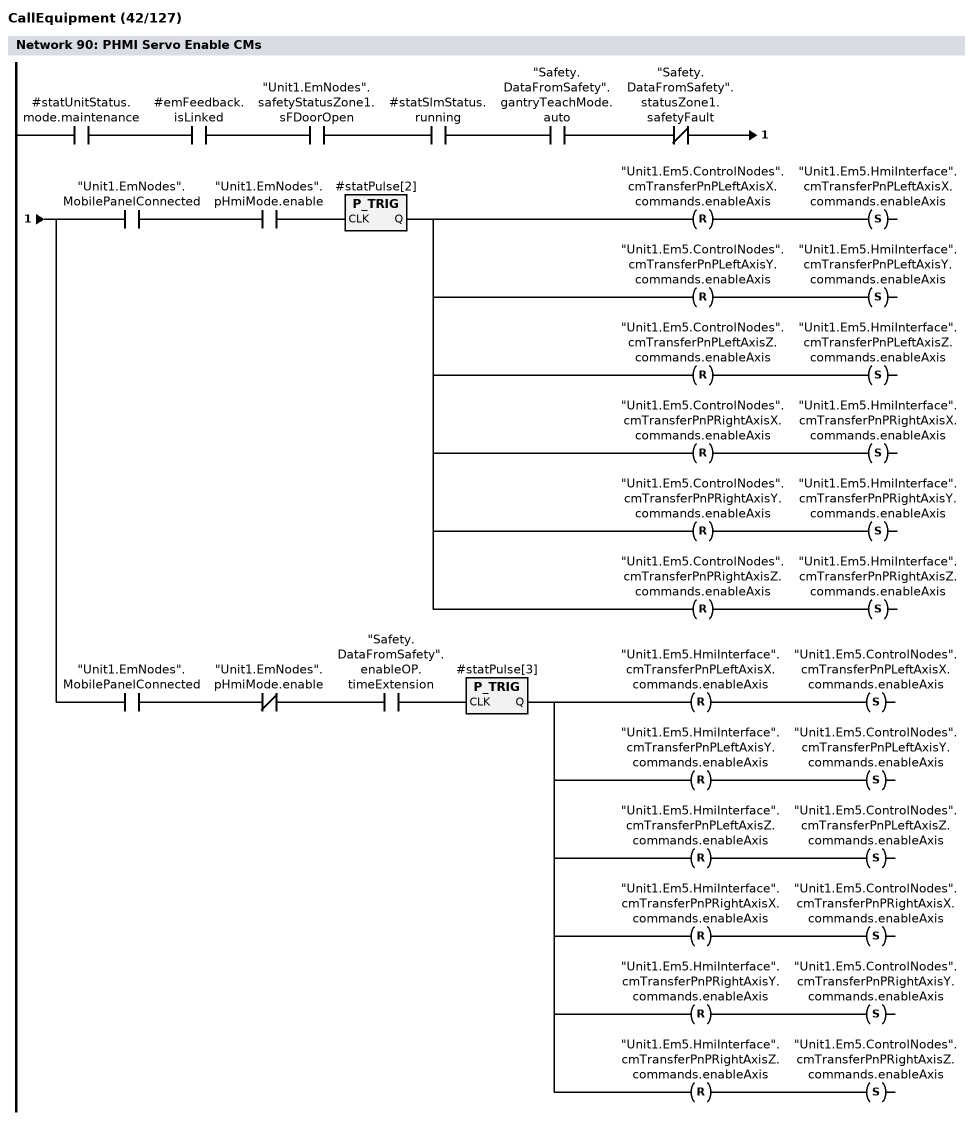
   RUNG wire#powerrail
      Contact( #statUnitStatus.mode.maintenance )
      Contact( #emFeedback.isLinked )
      Contact( "Unit1.EmNodes".safetyStatusZone1.sFDoorOpen )
      Contact( #statSlmStatus.running )
      Contact( "Safety.DataFromSafety".gantryTeachMode.auto )
      I_Contact( "Safety.DataFromSafety".statusZone1.safetyFault )
      wire#w1
      Contact( "Unit1.EmNodes".MobilePanelConnected )
      Contact( "Unit1.EmNodes".pHmiMode.enable )
      P_Trig( #statPulse[2] )
      wire#w2
      R_Coil( "Unit1.Em5.ControlNodes".cmTransferPnPLeftAxisX.commands.enableAxis )
      S_Coil( "Unit1.Em5.HmiInterface".cmTransferPnPLeftAxisX.commands.enableAxis )
   END_RUNG
   RUNG wire#w2
      R_Coil( "Unit1.Em5.ControlNodes".cmTransferPnPLeftAxisY.commands.enableAxis )
      S_Coil( "Unit1.Em5.HmiInterface".cmTransferPnPLeftAxisY.commands.enableAxis )
   END_RUNG
   RUNG wire#w2
      R_Coil( "Unit1.Em5.ControlNodes".cmTransferPnPLeftAxisZ.commands.enableAxis )
      S_Coil( "Unit1.Em5.HmiInterface".cmTransferPnPLeftAxisZ.commands.enableAxis )
   END_RUNG
   RUNG wire#w2
      R_Coil( "Unit1.Em5.ControlNodes".cmTransferPnPRightAxisX.commands.enableAxis )
      S_Coil( "Unit1.Em5.HmiInterface".cmTransferPnPRightAxisX.commands.enableAxis )
   END_RUNG
   RUNG wire#w2
      R_Coil( "Unit1.Em5.ControlNodes".cmTransferPnPRightAxisY.commands.enableAxis )
      S_Coil( "Unit1.Em5.HmiInterface".cmTransferPnPRightAxisY.commands.enableAxis )
   END_RUNG
   RUNG wire#w2
      R_Coil( "Unit1.Em5.ControlNodes".cmTransferPnPRightAxisZ.commands.enableAxis )
      S_Coil( "Unit1.Em5.HmiInterface".cmTransferPnPRightAxisZ.commands.enableAxis )
   END_RUNG
   RUNG wire#w1
      Contact( "Unit1.EmNodes".MobilePanelConnected )
      I_Contact( "Unit1.EmNodes".pHmiMode.enable )
      Contact( "Safety.DataFromSafety".enableOP.timeExtension )
      P_Trig( #statPulse[3] )
      wire#w3
      R_Coil( "Unit1.Em5.HmiInterface".cmTransferPnPLeftAxisX.commands.enableAxis )
      S_Coil( "Unit1.Em5.ControlNodes".cmTransferPnPLeftAxisX.commands.enableAxis )
   END_RUNG
   RUNG wire#w3
      R_Coil( "Unit1.Em5.HmiInterface".cmTransferPnPLeftAxisY.commands.enableAxis )
      S_Coil( "Unit1.Em5.ControlNodes".cmTransferPnPLeftAxisY.commands.enableAxis )
   END_RUNG
   RUNG wire#w3
      R_Coil( "Unit1.Em5.HmiInterface".cmTransferPnPLeftAxisZ.commands.enableAxis )
      S_Coil( "Unit1.Em5.ControlNodes".cmTransferPnPLeftAxisZ.commands.enableAxis )
   END_RUNG
   RUNG wire#w3
      R_Coil( "Unit1.Em5.HmiInterface".cmTransferPnPRightAxisX.commands.enableAxis )
      S_Coil( "Unit1.Em5.ControlNodes".cmTransferPnPRightAxisX.commands.enableAxis )
   END_RUNG
   RUNG wire#w3
      R_Coil( "Unit1.Em5.HmiInterface".cmTransferPnPRightAxisY.commands.enableAxis )
      S_Coil( "Unit1.Em5.ControlNodes".cmTransferPnPRightAxisY.commands.enableAxis )
   END_RUNG
   RUNG wire#w3
      R_Coil( "Unit1.Em5.HmiInterface".cmTransferPnPRightAxisZ.commands.enableAxis )
      S_Coil( "Unit1.Em5.ControlNodes".cmTransferPnPRightAxisZ.commands.enableAxis )
   END_RUNG
   // the same network as SCL:
   #_w1 := #statUnitStatus.mode.maintenance AND #emFeedback.isLinked AND "Unit1.EmNodes".safetyStatusZone1.sFDoorOpen AND #statSlmStatus.running AND "Safety.DataFromSafety".gantryTeachMode.auto AND NOT "Safety.DataFromSafety".statusZone1.safetyFault;
   #_w2 := #_w1 AND "Unit1.EmNodes".MobilePanelConnected AND "Unit1.EmNodes".pHmiMode.enable;
   #_w3 := #_w2 AND NOT #statPulse[2];   // rising edge
   #statPulse[2] := #_w2;
   IF #_w3 THEN
       "Unit1.Em5.ControlNodes".cmTransferPnPLeftAxisX.commands.enableAxis := FALSE;
       "Unit1.Em5.HmiInterface".cmTransferPnPLeftAxisX.commands.enableAxis := TRUE;
       "Unit1.Em5.ControlNodes".cmTransferPnPLeftAxisY.commands.enableAxis := FALSE;
       "Unit1.Em5.HmiInterface".cmTransferPnPLeftAxisY.commands.enableAxis := TRUE;
       "Unit1.Em5.ControlNodes".cmTransferPnPLeftAxisZ.commands.enableAxis := FALSE;
       "Unit1.Em5.HmiInterface".cmTransferPnPLeftAxisZ.commands.enableAxis := TRUE;
       "Unit1.Em5.ControlNodes".cmTransferPnPRightAxisX.commands.enableAxis := FALSE;
       "Unit1.Em5.HmiInterface".cmTransferPnPRightAxisX.commands.enableAxis := TRUE;
       "Unit1.Em5.ControlNodes".cmTransferPnPRightAxisY.commands.enableAxis := FALSE;
       "Unit1.Em5.HmiInterface".cmTransferPnPRightAxisY.commands.enableAxis := TRUE;
       "Unit1.Em5.ControlNodes".cmTransferPnPRightAxisZ.commands.enableAxis := FALSE;
       "Unit1.Em5.HmiInterface".cmTransferPnPRightAxisZ.commands.enableAxis := TRUE;
   END_IF;
   #_w4 := #_w1 AND "Unit1.EmNodes".MobilePanelConnected AND NOT "Unit1.EmNodes".pHmiMode.enable AND "Safety.DataFromSafety".enableOP.timeExtension;
   #_w5 := #_w4 AND NOT #statPulse[3];   // rising edge
   #statPulse[3] := #_w4;
   IF #_w5 THEN
       "Unit1.Em5.HmiInterface".cmTransferPnPLeftAxisX.commands.enableAxis := FALSE;
       "Unit1.Em5.ControlNodes".cmTransferPnPLeftAxisX.commands.enableAxis := TRUE;
       "Unit1.Em5.HmiInterface".cmTransferPnPLeftAxisY.commands.enableAxis := FALSE;
       "Unit1.Em5.ControlNodes".cmTransferPnPLeftAxisY.commands.enableAxis := TRUE;
       "Unit1.Em5.HmiInterface".cmTransferPnPLeftAxisZ.commands.enableAxis := FALSE;
       "Unit1.Em5.ControlNodes".cmTransferPnPLeftAxisZ.commands.enableAxis := TRUE;
       "Unit1.Em5.HmiInterface".cmTransferPnPRightAxisX.commands.enableAxis := FALSE;
       "Unit1.Em5.ControlNodes".cmTransferPnPRightAxisX.commands.enableAxis := TRUE;
       "Unit1.Em5.HmiInterface".cmTransferPnPRightAxisY.commands.enableAxis := FALSE;
       "Unit1.Em5.ControlNodes".cmTransferPnPRightAxisY.commands.enableAxis := TRUE;
       "Unit1.Em5.HmiInterface".cmTransferPnPRightAxisZ.commands.enableAxis := FALSE;
       "Unit1.Em5.ControlNodes".cmTransferPnPRightAxisZ.commands.enableAxis := TRUE;
   END_IF;
END_REGION

REGION Network 91: Sleep Mode Enable
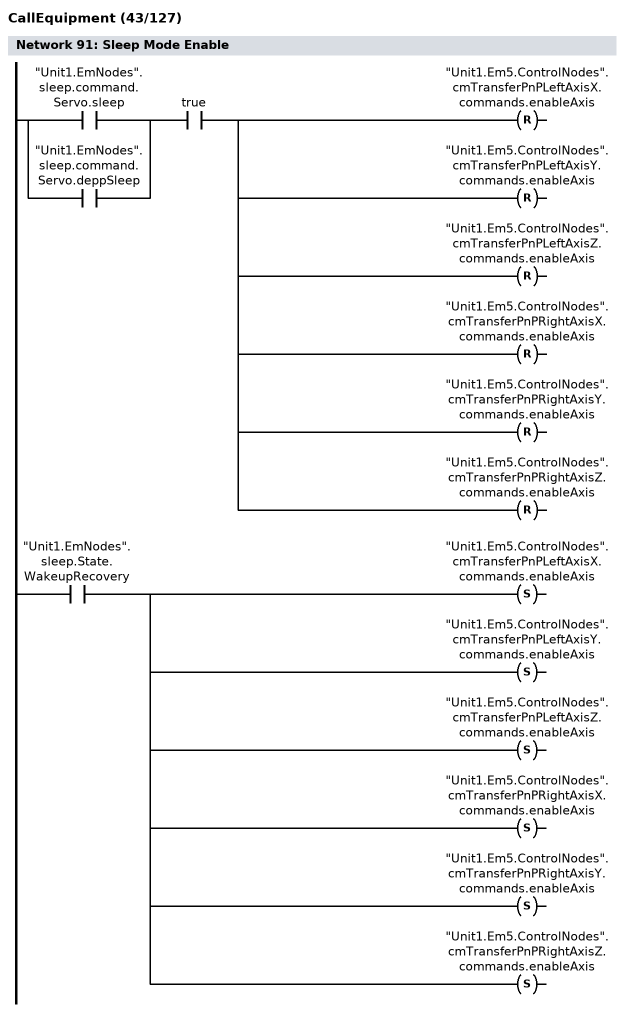
   RUNG wire#powerrail
      Contact( "Unit1.EmNodes".sleep.command.Servo.sleep )
      wire#w1
      Contact( true )
      wire#w2
      R_Coil( "Unit1.Em5.ControlNodes".cmTransferPnPLeftAxisX.commands.enableAxis )
   END_RUNG
   RUNG wire#powerrail
      Contact( "Unit1.EmNodes".sleep.command.Servo.deppSleep )
   END_RUNG wire#w1
   RUNG wire#w2
      R_Coil( "Unit1.Em5.ControlNodes".cmTransferPnPLeftAxisY.commands.enableAxis )
   END_RUNG
   RUNG wire#w2
      R_Coil( "Unit1.Em5.ControlNodes".cmTransferPnPLeftAxisZ.commands.enableAxis )
   END_RUNG
   RUNG wire#w2
      R_Coil( "Unit1.Em5.ControlNodes".cmTransferPnPRightAxisX.commands.enableAxis )
   END_RUNG
   RUNG wire#w2
      R_Coil( "Unit1.Em5.ControlNodes".cmTransferPnPRightAxisY.commands.enableAxis )
   END_RUNG
   RUNG wire#w2
      R_Coil( "Unit1.Em5.ControlNodes".cmTransferPnPRightAxisZ.commands.enableAxis )
   END_RUNG
   RUNG wire#powerrail
      Contact( "Unit1.EmNodes".sleep.State.WakeupRecovery )
      wire#w3
      S_Coil( "Unit1.Em5.ControlNodes".cmTransferPnPLeftAxisX.commands.enableAxis )
   END_RUNG
   RUNG wire#w3
      S_Coil( "Unit1.Em5.ControlNodes".cmTransferPnPLeftAxisY.commands.enableAxis )
   END_RUNG
   RUNG wire#w3
      S_Coil( "Unit1.Em5.ControlNodes".cmTransferPnPLeftAxisZ.commands.enableAxis )
   END_RUNG
   RUNG wire#w3
      S_Coil( "Unit1.Em5.ControlNodes".cmTransferPnPRightAxisX.commands.enableAxis )
   END_RUNG
   RUNG wire#w3
      S_Coil( "Unit1.Em5.ControlNodes".cmTransferPnPRightAxisY.commands.enableAxis )
   END_RUNG
   RUNG wire#w3
      S_Coil( "Unit1.Em5.ControlNodes".cmTransferPnPRightAxisZ.commands.enableAxis )
   END_RUNG
   // the same network as SCL:
   IF ("Unit1.EmNodes".sleep.command.Servo.sleep OR "Unit1.EmNodes".sleep.command.Servo.deppSleep) AND true THEN
       "Unit1.Em5.ControlNodes".cmTransferPnPLeftAxisX.commands.enableAxis := FALSE;
       "Unit1.Em5.ControlNodes".cmTransferPnPLeftAxisY.commands.enableAxis := FALSE;
       "Unit1.Em5.ControlNodes".cmTransferPnPLeftAxisZ.commands.enableAxis := FALSE;
       "Unit1.Em5.ControlNodes".cmTransferPnPRightAxisX.commands.enableAxis := FALSE;
       "Unit1.Em5.ControlNodes".cmTransferPnPRightAxisY.commands.enableAxis := FALSE;
       "Unit1.Em5.ControlNodes".cmTransferPnPRightAxisZ.commands.enableAxis := FALSE;
   END_IF;
   IF "Unit1.EmNodes".sleep.State.WakeupRecovery THEN
       "Unit1.Em5.ControlNodes".cmTransferPnPLeftAxisX.commands.enableAxis := TRUE;
       "Unit1.Em5.ControlNodes".cmTransferPnPLeftAxisY.commands.enableAxis := TRUE;
       "Unit1.Em5.ControlNodes".cmTransferPnPLeftAxisZ.commands.enableAxis := TRUE;
       "Unit1.Em5.ControlNodes".cmTransferPnPRightAxisX.commands.enableAxis := TRUE;
       "Unit1.Em5.ControlNodes".cmTransferPnPRightAxisY.commands.enableAxis := TRUE;
       "Unit1.Em5.ControlNodes".cmTransferPnPRightAxisZ.commands.enableAxis := TRUE;
   END_IF;
END_REGION

REGION Network 92: LBC_Axis64Pos Operation Mode
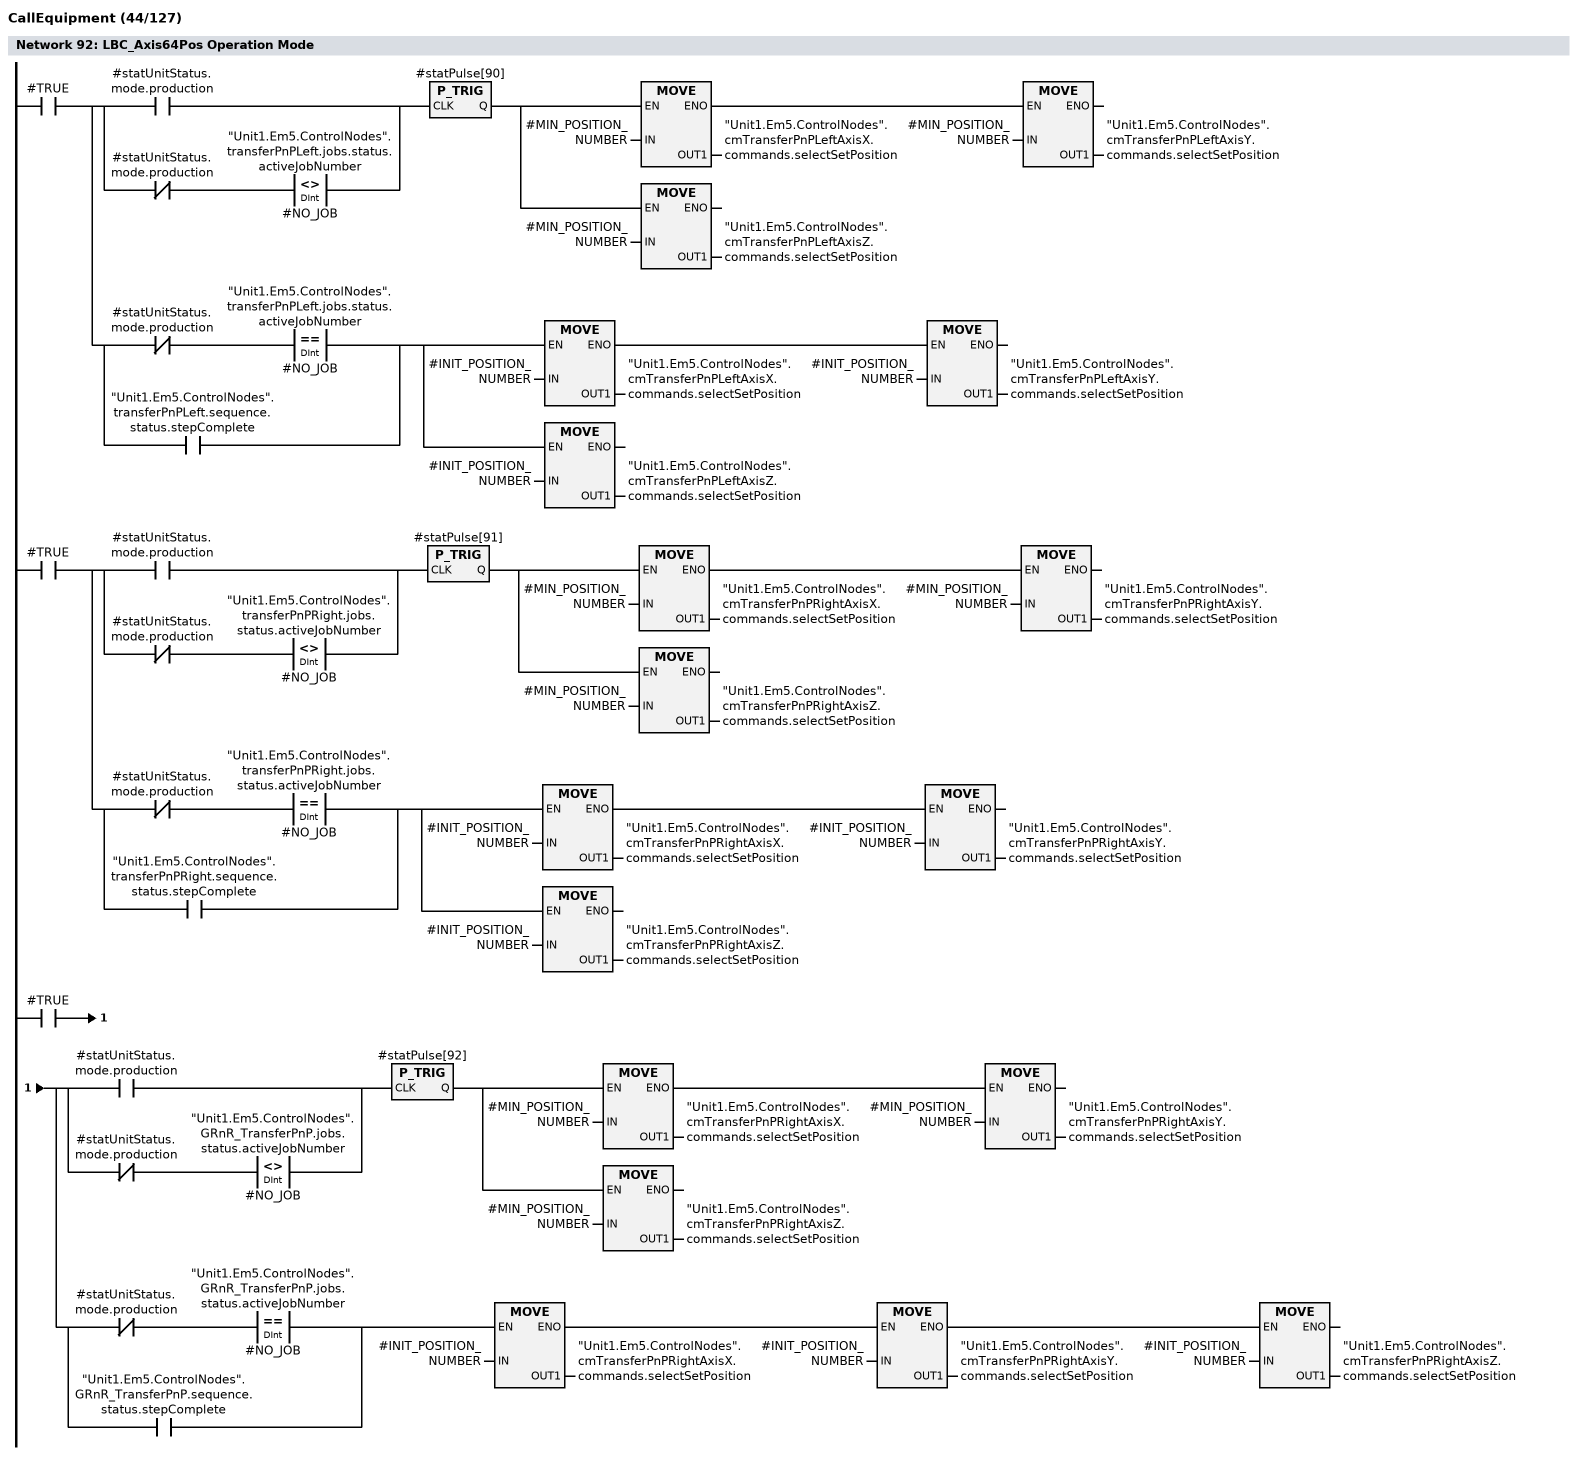
   RUNG wire#powerrail
      Contact( #TRUE )
      wire#w1
      Contact( #statUnitStatus.mode.production )
      wire#w2
      P_Trig( #statPulse[90] )
      wire#w3
      Move(in := #MIN_POSITION_NUMBER, out1 => "Unit1.Em5.ControlNodes".cmTransferPnPLeftAxisX.commands.selectSetPosition)
      Move(in := #MIN_POSITION_NUMBER, out1 => "Unit1.Em5.ControlNodes".cmTransferPnPLeftAxisY.commands.selectSetPosition)
   END_RUNG
   RUNG wire#w1
      I_Contact( #statUnitStatus.mode.production )
      { S7_Templates := "SrcType := DInt" } NE_Contact(in1 := "Unit1.Em5.ControlNodes".transferPnPLeft.jobs.status.activeJobNumber, in2 := #NO_JOB)
   END_RUNG wire#w2
   RUNG wire#w3
      Move(in := #MIN_POSITION_NUMBER, out1 => "Unit1.Em5.ControlNodes".cmTransferPnPLeftAxisZ.commands.selectSetPosition)
   END_RUNG
   RUNG wire#w1
      I_Contact( #statUnitStatus.mode.production )
      { S7_Templates := "SrcType := DInt" } EQ_Contact(in1 := "Unit1.Em5.ControlNodes".transferPnPLeft.jobs.status.activeJobNumber, in2 := #NO_JOB)
      wire#w4
      Move(in := #INIT_POSITION_NUMBER, out1 => "Unit1.Em5.ControlNodes".cmTransferPnPLeftAxisX.commands.selectSetPosition)
      Move(in := #INIT_POSITION_NUMBER, out1 => "Unit1.Em5.ControlNodes".cmTransferPnPLeftAxisY.commands.selectSetPosition)
   END_RUNG
   RUNG wire#w1
      Contact( "Unit1.Em5.ControlNodes".transferPnPLeft.sequence.status.stepComplete )
   END_RUNG wire#w4
   RUNG wire#w4
      Move(in := #INIT_POSITION_NUMBER, out1 => "Unit1.Em5.ControlNodes".cmTransferPnPLeftAxisZ.commands.selectSetPosition)
   END_RUNG
   RUNG wire#powerrail
      Contact( #TRUE )
      wire#w5
      Contact( #statUnitStatus.mode.production )
      wire#w6
      P_Trig( #statPulse[91] )
      wire#w7
      Move(in := #MIN_POSITION_NUMBER, out1 => "Unit1.Em5.ControlNodes".cmTransferPnPRightAxisX.commands.selectSetPosition)
      Move(in := #MIN_POSITION_NUMBER, out1 => "Unit1.Em5.ControlNodes".cmTransferPnPRightAxisY.commands.selectSetPosition)
   END_RUNG
   RUNG wire#w5
      I_Contact( #statUnitStatus.mode.production )
      { S7_Templates := "SrcType := DInt" } NE_Contact(in1 := "Unit1.Em5.ControlNodes".transferPnPRight.jobs.status.activeJobNumber, in2 := #NO_JOB)
   END_RUNG wire#w6
   RUNG wire#w7
      Move(in := #MIN_POSITION_NUMBER, out1 => "Unit1.Em5.ControlNodes".cmTransferPnPRightAxisZ.commands.selectSetPosition)
   END_RUNG
   RUNG wire#w5
      I_Contact( #statUnitStatus.mode.production )
      { S7_Templates := "SrcType := DInt" } EQ_Contact(in1 := "Unit1.Em5.ControlNodes".transferPnPRight.jobs.status.activeJobNumber, in2 := #NO_JOB)
      wire#w8
      Move(in := #INIT_POSITION_NUMBER, out1 => "Unit1.Em5.ControlNodes".cmTransferPnPRightAxisX.commands.selectSetPosition)
      Move(in := #INIT_POSITION_NUMBER, out1 => "Unit1.Em5.ControlNodes".cmTransferPnPRightAxisY.commands.selectSetPosition)
   END_RUNG
   RUNG wire#w5
      Contact( "Unit1.Em5.ControlNodes".transferPnPRight.sequence.status.stepComplete )
   END_RUNG wire#w8
   RUNG wire#w8
      Move(in := #INIT_POSITION_NUMBER, out1 => "Unit1.Em5.ControlNodes".cmTransferPnPRightAxisZ.commands.selectSetPosition)
   END_RUNG
   RUNG wire#powerrail
      Contact( #TRUE )
      wire#w9
      Contact( #statUnitStatus.mode.production )
      wire#w10
      P_Trig( #statPulse[92] )
      wire#w11
      Move(in := #MIN_POSITION_NUMBER, out1 => "Unit1.Em5.ControlNodes".cmTransferPnPRightAxisX.commands.selectSetPosition)
      Move(in := #MIN_POSITION_NUMBER, out1 => "Unit1.Em5.ControlNodes".cmTransferPnPRightAxisY.commands.selectSetPosition)
   END_RUNG
   RUNG wire#w9
      I_Contact( #statUnitStatus.mode.production )
      { S7_Templates := "SrcType := DInt" } NE_Contact(in1 := "Unit1.Em5.ControlNodes".GRnR_TransferPnP.jobs.status.activeJobNumber, in2 := #NO_JOB)
   END_RUNG wire#w10
   RUNG wire#w11
      Move(in := #MIN_POSITION_NUMBER, out1 => "Unit1.Em5.ControlNodes".cmTransferPnPRightAxisZ.commands.selectSetPosition)
   END_RUNG
   RUNG wire#w9
      I_Contact( #statUnitStatus.mode.production )
      { S7_Templates := "SrcType := DInt" } EQ_Contact(in1 := "Unit1.Em5.ControlNodes".GRnR_TransferPnP.jobs.status.activeJobNumber, in2 := #NO_JOB)
      wire#w12
      Move(in := #INIT_POSITION_NUMBER, out1 => "Unit1.Em5.ControlNodes".cmTransferPnPRightAxisX.commands.selectSetPosition)
      Move(in := #INIT_POSITION_NUMBER, out1 => "Unit1.Em5.ControlNodes".cmTransferPnPRightAxisY.commands.selectSetPosition)
      Move(in := #INIT_POSITION_NUMBER, out1 => "Unit1.Em5.ControlNodes".cmTransferPnPRightAxisZ.commands.selectSetPosition)
   END_RUNG
   RUNG wire#w9
      Contact( "Unit1.Em5.ControlNodes".GRnR_TransferPnP.sequence.status.stepComplete )
   END_RUNG wire#w12
   // the same network as SCL:
   #_w1 := #TRUE AND (#statUnitStatus.mode.production OR (NOT #statUnitStatus.mode.production AND ("Unit1.Em5.ControlNodes".transferPnPLeft.jobs.status.activeJobNumber <> #NO_JOB)));
   #_w2 := #_w1 AND NOT #statPulse[90];   // rising edge
   #statPulse[90] := #_w1;
   IF #_w2 THEN
       "Unit1.Em5.ControlNodes".cmTransferPnPLeftAxisX.commands.selectSetPosition := #MIN_POSITION_NUMBER;
       "Unit1.Em5.ControlNodes".cmTransferPnPLeftAxisY.commands.selectSetPosition := #MIN_POSITION_NUMBER;
       "Unit1.Em5.ControlNodes".cmTransferPnPLeftAxisZ.commands.selectSetPosition := #MIN_POSITION_NUMBER;
   END_IF;
   IF #TRUE AND ((NOT #statUnitStatus.mode.production AND ("Unit1.Em5.ControlNodes".transferPnPLeft.jobs.status.activeJobNumber = #NO_JOB)) OR "Unit1.Em5.ControlNodes".transferPnPLeft.sequence.status.stepComplete) THEN
       "Unit1.Em5.ControlNodes".cmTransferPnPLeftAxisX.commands.selectSetPosition := #INIT_POSITION_NUMBER;
       "Unit1.Em5.ControlNodes".cmTransferPnPLeftAxisY.commands.selectSetPosition := #INIT_POSITION_NUMBER;
       "Unit1.Em5.ControlNodes".cmTransferPnPLeftAxisZ.commands.selectSetPosition := #INIT_POSITION_NUMBER;
   END_IF;
   #_w3 := #TRUE AND (#statUnitStatus.mode.production OR (NOT #statUnitStatus.mode.production AND ("Unit1.Em5.ControlNodes".transferPnPRight.jobs.status.activeJobNumber <> #NO_JOB)));
   #_w4 := #_w3 AND NOT #statPulse[91];   // rising edge
   #statPulse[91] := #_w3;
   IF #_w4 THEN
       "Unit1.Em5.ControlNodes".cmTransferPnPRightAxisX.commands.selectSetPosition := #MIN_POSITION_NUMBER;
       "Unit1.Em5.ControlNodes".cmTransferPnPRightAxisY.commands.selectSetPosition := #MIN_POSITION_NUMBER;
       "Unit1.Em5.ControlNodes".cmTransferPnPRightAxisZ.commands.selectSetPosition := #MIN_POSITION_NUMBER;
   END_IF;
   IF #TRUE AND ((NOT #statUnitStatus.mode.production AND ("Unit1.Em5.ControlNodes".transferPnPRight.jobs.status.activeJobNumber = #NO_JOB)) OR "Unit1.Em5.ControlNodes".transferPnPRight.sequence.status.stepComplete) THEN
       "Unit1.Em5.ControlNodes".cmTransferPnPRightAxisX.commands.selectSetPosition := #INIT_POSITION_NUMBER;
       "Unit1.Em5.ControlNodes".cmTransferPnPRightAxisY.commands.selectSetPosition := #INIT_POSITION_NUMBER;
       "Unit1.Em5.ControlNodes".cmTransferPnPRightAxisZ.commands.selectSetPosition := #INIT_POSITION_NUMBER;
   END_IF;
   #_w5 := #TRUE AND (#statUnitStatus.mode.production OR (NOT #statUnitStatus.mode.production AND ("Unit1.Em5.ControlNodes".GRnR_TransferPnP.jobs.status.activeJobNumber <> #NO_JOB)));
   #_w6 := #_w5 AND NOT #statPulse[92];   // rising edge
   #statPulse[92] := #_w5;
   IF #_w6 THEN
       "Unit1.Em5.ControlNodes".cmTransferPnPRightAxisX.commands.selectSetPosition := #MIN_POSITION_NUMBER;
       "Unit1.Em5.ControlNodes".cmTransferPnPRightAxisY.commands.selectSetPosition := #MIN_POSITION_NUMBER;
       "Unit1.Em5.ControlNodes".cmTransferPnPRightAxisZ.commands.selectSetPosition := #MIN_POSITION_NUMBER;
   END_IF;
   IF #TRUE AND ((NOT #statUnitStatus.mode.production AND ("Unit1.Em5.ControlNodes".GRnR_TransferPnP.jobs.status.activeJobNumber = #NO_JOB)) OR "Unit1.Em5.ControlNodes".GRnR_TransferPnP.sequence.status.stepComplete) THEN
       "Unit1.Em5.ControlNodes".cmTransferPnPRightAxisX.commands.selectSetPosition := #INIT_POSITION_NUMBER;
       "Unit1.Em5.ControlNodes".cmTransferPnPRightAxisY.commands.selectSetPosition := #INIT_POSITION_NUMBER;
       "Unit1.Em5.ControlNodes".cmTransferPnPRightAxisZ.commands.selectSetPosition := #INIT_POSITION_NUMBER;
   END_IF;
END_REGION

REGION Network 93: Production Mode Change -> Servo Stop
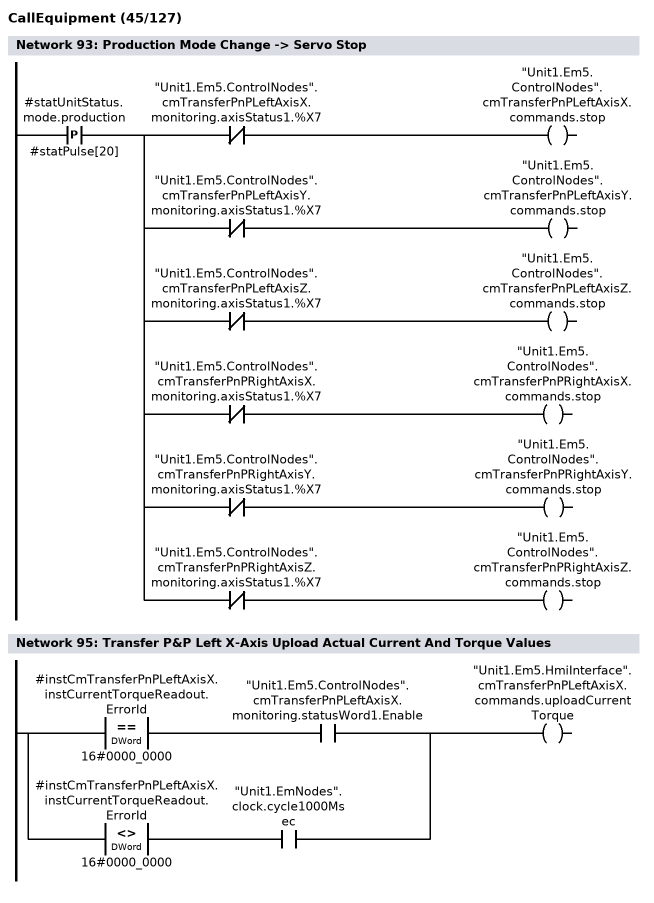
   RUNG wire#powerrail
      P_Contact(operand := #statUnitStatus.mode.production, bit := #statPulse[20])
      wire#w1
      I_Contact( "Unit1.Em5.ControlNodes".cmTransferPnPLeftAxisX.monitoring.axisStatus1.%X7 )
      Coil( "Unit1.Em5.ControlNodes".cmTransferPnPLeftAxisX.commands.stop )
   END_RUNG
   RUNG wire#w1
      I_Contact( "Unit1.Em5.ControlNodes".cmTransferPnPLeftAxisY.monitoring.axisStatus1.%X7 )
      Coil( "Unit1.Em5.ControlNodes".cmTransferPnPLeftAxisY.commands.stop )
   END_RUNG
   RUNG wire#w1
      I_Contact( "Unit1.Em5.ControlNodes".cmTransferPnPLeftAxisZ.monitoring.axisStatus1.%X7 )
      Coil( "Unit1.Em5.ControlNodes".cmTransferPnPLeftAxisZ.commands.stop )
   END_RUNG
   RUNG wire#w1
      I_Contact( "Unit1.Em5.ControlNodes".cmTransferPnPRightAxisX.monitoring.axisStatus1.%X7 )
      Coil( "Unit1.Em5.ControlNodes".cmTransferPnPRightAxisX.commands.stop )
   END_RUNG
   RUNG wire#w1
      I_Contact( "Unit1.Em5.ControlNodes".cmTransferPnPRightAxisY.monitoring.axisStatus1.%X7 )
      Coil( "Unit1.Em5.ControlNodes".cmTransferPnPRightAxisY.commands.stop )
   END_RUNG
   RUNG wire#w1
      I_Contact( "Unit1.Em5.ControlNodes".cmTransferPnPRightAxisZ.monitoring.axisStatus1.%X7 )
      Coil( "Unit1.Em5.ControlNodes".cmTransferPnPRightAxisZ.commands.stop )
   END_RUNG
   // the same network as SCL:
   #_w1 := #statUnitStatus.mode.production AND NOT #statPulse[20];   // rising edge of #statUnitStatus.mode.production
   #statPulse[20] := #statUnitStatus.mode.production;
   "Unit1.Em5.ControlNodes".cmTransferPnPLeftAxisX.commands.stop := #_w1 AND NOT "Unit1.Em5.ControlNodes".cmTransferPnPLeftAxisX.monitoring.axisStatus1.%X7;
   "Unit1.Em5.ControlNodes".cmTransferPnPLeftAxisY.commands.stop := #_w1 AND NOT "Unit1.Em5.ControlNodes".cmTransferPnPLeftAxisY.monitoring.axisStatus1.%X7;
   "Unit1.Em5.ControlNodes".cmTransferPnPLeftAxisZ.commands.stop := #_w1 AND NOT "Unit1.Em5.ControlNodes".cmTransferPnPLeftAxisZ.monitoring.axisStatus1.%X7;
   "Unit1.Em5.ControlNodes".cmTransferPnPRightAxisX.commands.stop := #_w1 AND NOT "Unit1.Em5.ControlNodes".cmTransferPnPRightAxisX.monitoring.axisStatus1.%X7;
   "Unit1.Em5.ControlNodes".cmTransferPnPRightAxisY.commands.stop := #_w1 AND NOT "Unit1.Em5.ControlNodes".cmTransferPnPRightAxisY.monitoring.axisStatus1.%X7;
   "Unit1.Em5.ControlNodes".cmTransferPnPRightAxisZ.commands.stop := #_w1 AND NOT "Unit1.Em5.ControlNodes".cmTransferPnPRightAxisZ.monitoring.axisStatus1.%X7;
END_REGION

REGION Network 95: Transfer P&P Left X-Axis Upload Actual Current And Torque Values
   RUNG wire#powerrail
      { S7_Templates := "SrcType := DWord" } EQ_Contact(in1 := #instCmTransferPnPLeftAxisX.instCurrentTorqueReadout.ErrorId, in2 := 16#0000_0000)
      Contact( "Unit1.Em5.ControlNodes".cmTransferPnPLeftAxisX.monitoring.statusWord1.Enable )
      wire#w1
      Coil( "Unit1.Em5.HmiInterface".cmTransferPnPLeftAxisX.commands.uploadCurrentTorque )
   END_RUNG
   RUNG wire#powerrail
      { S7_Templates := "SrcType := DWord" } NE_Contact(in1 := #instCmTransferPnPLeftAxisX.instCurrentTorqueReadout.ErrorId, in2 := 16#0000_0000)
      Contact( "Unit1.EmNodes".clock.cycle1000Msec )
   END_RUNG wire#w1
   // the same network as SCL:
   "Unit1.Em5.HmiInterface".cmTransferPnPLeftAxisX.commands.uploadCurrentTorque := ((#instCmTransferPnPLeftAxisX.instCurrentTorqueReadout.ErrorId = 16#0000_0000) AND "Unit1.Em5.ControlNodes".cmTransferPnPLeftAxisX.monitoring.statusWord1.Enable) OR ((#instCmTransferPnPLeftAxisX.instCurrentTorqueReadout.ErrorId <> 16#0000_0000) AND "Unit1.EmNodes".clock.cycle1000Msec);
END_REGION

